(* IEC 61131-3 sources: SmartHomeNew/snapshots/2026-05-19 (part 4) *)

(* ---- FB_Water_Runtime_Hardening.st ---- *)
FUNCTION_BLOCK FB_Water_Runtime_Hardening
VAR_INPUT
    VI_Enable : BOOL;
    VI_System_Time_MS : UDINT;
END_VAR
VAR
    L_i : INT;

    L_FSM : ST_Water_Recovery_FSM_State;
    L_Event : ST_Water_Event_Log_Record;

    L_Empty_FSM : ST_Water_Recovery_FSM_State;
    L_Empty_Event : ST_Water_Event_Log_Record;

    L_Any_Rollback : BOOL;
    L_Any_Escalation : BOOL;
END_VAR

IF NOT VI_Enable THEN
    GVL_Water_Runtime_Hardening.G_Runtime_Valid := FALSE;
    RETURN;
END_IF;

L_Any_Rollback := FALSE;
L_Any_Escalation := FALSE;

FOR L_i := 1 TO GVL_CONSTANTS.C_MAX_FLOOD_SENSORS DO

    // Recovery FSM.
    L_FSM := L_Empty_FSM;
    L_FSM.Runtime_Valid := TRUE;

    L_FSM.Runtime_System_Time_MS :=
        VI_System_Time_MS;

    L_FSM.Recovery_Domain_Id :=
        GVL_Water_Topology_Config.G_Config_Record[L_i].Recovery_Domain_Id;

    L_FSM.Recovery_Requested :=
        GVL_INTENT_SAFETY.I_Water_Selective_Recovery_Allowed;

    L_FSM.Recovery_Sequencing_Active :=
        GVL_Water_Orchestration.G_Orchestration_State[L_i].Recovery_Sequence_Active;

    L_FSM.Recovery_Verification_Window_Active :=
        GVL_Water_Orchestration.G_Orchestration_State[L_i].Observation_Window_Active;

    // Conservative runtime hardening.
    IF GVL_Water_Physical_Runtime.G_Convergence_State[L_i].Escalation_Required THEN

        L_FSM.Rollback_Required := TRUE;
        L_FSM.Escalation_Required := TRUE;
        L_FSM.Operator_Ack_Required := TRUE;
        L_FSM.Recovery_Denied := TRUE;
        L_FSM.FSM_State := 100;

        L_FSM.Status_Code := 2;
        L_FSM.Status_Text :=
            'Recovery rollback escalation active';

    ELSIF L_FSM.Recovery_Requested THEN

        L_FSM.Recovery_Completed := TRUE;
        L_FSM.FSM_State := 10;

        L_FSM.Status_Code := 1;
        L_FSM.Status_Text :=
            'Recovery sequencing active';

    ELSE

        L_FSM.FSM_State := 0;

        L_FSM.Status_Code := 0;
        L_FSM.Status_Text :=
            'Recovery FSM idle';

    END_IF;

    GVL_Water_Runtime_Hardening.G_Recovery_FSM[L_i] :=
        L_FSM;

    // Runtime event publication.
    IF L_i <= 128 THEN

        L_Event := L_Empty_Event;
        L_Event.Runtime_Valid := TRUE;

        L_Event.Event_Time_MS := VI_System_Time_MS;
        L_Event.Event_Id := TO_UINT(L_i);

        IF L_FSM.Escalation_Required THEN
            L_Event.Event_Text :=
                'Water runtime escalation active';
        ELSE
            L_Event.Event_Text :=
                'Water runtime healthy';
        END_IF;

        GVL_Water_Runtime_Hardening.G_Event_Log[L_i] :=
            L_Event;

    END_IF;

    L_Any_Rollback :=
        L_Any_Rollback
        OR L_FSM.Rollback_Required;

    L_Any_Escalation :=
        L_Any_Escalation
        OR L_FSM.Escalation_Required;

END_FOR;

GVL_Water_Runtime_Hardening.G_Runtime_Quarantine_Active :=
    L_Any_Escalation;

GVL_Water_Runtime_Hardening.G_Service_Mode_Active := FALSE;
GVL_Water_Runtime_Hardening.G_Maintenance_Mode_Active := FALSE;

GVL_Water_Runtime_Hardening.G_Any_Rollback_Required :=
    L_Any_Rollback;

GVL_Water_Runtime_Hardening.G_Any_Escalation_Required :=
    L_Any_Escalation;

GVL_Water_Runtime_Hardening.G_Runtime_Valid := TRUE;
GVL_Water_Runtime_Hardening.G_Last_Update_MS := VI_System_Time_MS;

IF L_Any_Escalation THEN
    GVL_Water_Runtime_Hardening.G_Status_Code := 2;
    GVL_Water_Runtime_Hardening.G_Status_Text :=
        'Runtime quarantine escalation active';
ELSIF L_Any_Rollback THEN
    GVL_Water_Runtime_Hardening.G_Status_Code := 1;
    GVL_Water_Runtime_Hardening.G_Status_Text :=
        'Recovery rollback active';
ELSE
    GVL_Water_Runtime_Hardening.G_Status_Code := 0;
    GVL_Water_Runtime_Hardening.G_Status_Text :=
        'Production runtime hardening active';
END_IF;

END_FUNCTION_BLOCK

(* ---- FB_Water_Valve_Feedback_Runtime.st ---- *)
FUNCTION_BLOCK FB_Water_Valve_Feedback_Runtime
VAR_INPUT
    VI_Enable : BOOL;
    VI_System_Time_MS : UDINT;
END_VAR
VAR
    L_i : INT;

    L_Output : ST_Water_Output_Projection_State;
    L_State : ST_Water_Valve_Feedback_State;
    L_Empty_State : ST_Water_Valve_Feedback_State;

    L_Any_Degraded : BOOL;
    L_Any_Timeout : BOOL;
    L_Any_Conflict : BOOL;
END_VAR

IF NOT VI_Enable THEN
    GVL_Water_Valve_Feedback.G_Runtime_Valid := FALSE;
    RETURN;
END_IF;

L_Any_Degraded := FALSE;
L_Any_Timeout := FALSE;
L_Any_Conflict := FALSE;

FOR L_i := 1 TO GVL_CONSTANTS.C_MAX_FLOOD_SENSORS DO

    L_Output := GVL_Water_Output_Projection.G_Output_Projection_State[L_i];

    L_State := L_Empty_State;
    L_State.Runtime_Valid := TRUE;

    L_State.Runtime_System_Time_MS := VI_System_Time_MS;
    L_State.Valve_Group_Id := L_Output.Valve_Group_Id;

    // Feedback integration hook.
    // Conservative observe-only mode until physical DI binding is connected.
    L_State.Feedback_Available := FALSE;

    // No forced degraded state in observe-only mode.
    IF L_State.Feedback_Available THEN

        IF L_State.Physical_Open_Feedback
           AND L_State.Physical_Closed_Feedback THEN

            L_State.Feedback_Conflict := TRUE;
            L_State.Valve_Degraded := TRUE;

        END_IF;

        L_State.Confirmed_Open :=
            L_State.Physical_Open_Feedback
            AND NOT L_State.Physical_Closed_Feedback;

        L_State.Confirmed_Closed :=
            L_State.Physical_Closed_Feedback
            AND NOT L_State.Physical_Open_Feedback;

    ELSE

        L_State.Confirmation_Unknown := TRUE;

    END_IF;

    IF L_State.Feedback_Conflict THEN
        L_State.Status_Code := 3;
        L_State.Status_Text :=
            'Valve feedback conflict detected';
    ELSIF L_State.Feedback_Timeout THEN
        L_State.Status_Code := 2;
        L_State.Status_Text :=
            'Valve feedback timeout';
    ELSIF L_State.Confirmation_Unknown THEN
        L_State.Status_Code := 1;
        L_State.Status_Text :=
            'Valve feedback unavailable';
    ELSE
        L_State.Status_Code := 0;
        L_State.Status_Text :=
            'Valve feedback healthy';
    END_IF;

    GVL_Water_Valve_Feedback.G_Valve_Feedback_State[L_i] :=
        L_State;

    L_Any_Degraded :=
        L_Any_Degraded
        OR L_State.Valve_Degraded;

    L_Any_Timeout :=
        L_Any_Timeout
        OR L_State.Feedback_Timeout;

    L_Any_Conflict :=
        L_Any_Conflict
        OR L_State.Feedback_Conflict;

END_FOR;

GVL_Water_Valve_Feedback.G_Any_Degraded :=
    L_Any_Degraded;

GVL_Water_Valve_Feedback.G_Any_Timeout :=
    L_Any_Timeout;

GVL_Water_Valve_Feedback.G_Any_Conflict :=
    L_Any_Conflict;

GVL_Water_Valve_Feedback.G_Runtime_Valid := TRUE;
GVL_Water_Valve_Feedback.G_Last_Update_MS := VI_System_Time_MS;

IF L_Any_Conflict THEN
    GVL_Water_Valve_Feedback.G_Status_Code := 3;
    GVL_Water_Valve_Feedback.G_Status_Text :=
        'Valve feedback conflicts detected';
ELSIF L_Any_Timeout THEN
    GVL_Water_Valve_Feedback.G_Status_Code := 2;
    GVL_Water_Valve_Feedback.G_Status_Text :=
        'Valve feedback degraded';
ELSIF L_Any_Degraded THEN
    GVL_Water_Valve_Feedback.G_Status_Code := 1;
    GVL_Water_Valve_Feedback.G_Status_Text :=
        'Valve diagnostics degraded';
ELSE
    GVL_Water_Valve_Feedback.G_Status_Code := 0;
    GVL_Water_Valve_Feedback.G_Status_Text :=
        'Valve feedback runtime healthy';
END_IF;

END_FUNCTION_BLOCK

(* ---- FB_Water_Valve_Runtime_Governance.st ---- *)
FUNCTION_BLOCK FB_Water_Valve_Runtime_Governance
VAR_INPUT
    VI_Enable : BOOL;
    VI_System_Time_MS : UDINT;
END_VAR
VAR
    L_i : INT;

    L_Authority : ST_Water_Isolation_Authority_State;
    L_Valve : ST_Water_Valve_Runtime_State;
    L_Empty_Valve : ST_Water_Valve_Runtime_State;

    L_Any_Degraded : BOOL;
    L_Any_Confirmation_Unknown : BOOL;
    L_Any_Unsafe_Reopen : BOOL;
END_VAR

IF NOT VI_Enable THEN
    GVL_Water_Valve_Runtime.G_Runtime_Valid := FALSE;
    RETURN;
END_IF;

L_Any_Degraded := FALSE;
L_Any_Confirmation_Unknown := FALSE;
L_Any_Unsafe_Reopen := FALSE;

FOR L_i := 1 TO GVL_CONSTANTS.C_MAX_FLOOD_SENSORS DO

    L_Authority :=
        GVL_Water_Isolation_Authority.G_Authority_State[L_i];

    L_Valve := L_Empty_Valve;
    L_Valve.Runtime_Valid := TRUE;

    L_Valve.Runtime_System_Time_MS := VI_System_Time_MS;

    L_Valve.Valve_Id := L_Authority.Valve_Group_Id;
    L_Valve.Valve_Group_Id := L_Authority.Valve_Group_Id;

    L_Valve.Close_Requested :=
        L_Authority.Selective_Authority_Allowed
        OR L_Authority.Global_Fallback_Required;

    L_Valve.Global_Fallback_Request :=
        L_Authority.Global_Fallback_Required;

    L_Valve.Selective_Authority_Allowed :=
        L_Authority.Selective_Authority_Allowed;

    // Observe-only compatibility visibility.
    L_Valve.Physical_Output_Active :=
        GVL_COMMAND_SHADOW.G_Close_Valve_35
        OR GVL_COMMAND_SHADOW.G_Close_Valve_36;

    L_Valve.Output_Command_Projected :=
        L_Valve.Close_Requested;

    // Feedback/runtime hooks.
    L_Valve.Confirmation_Available :=
        GVL_Water_Valve_Feedback.G_Valve_Feedback_State[L_i].Feedback_Available;

    IF L_Valve.Confirmation_Available THEN

        L_Valve.Confirmed_Closed :=
            GVL_Water_Valve_Feedback.G_Valve_Feedback_State[L_i].Confirmed_Closed;

    ELSE

        L_Valve.Confirmation_Unknown := TRUE;

    END_IF;

    // Observe-only semantics must not force degraded state.
    L_Valve.Diagnostics_Available := FALSE;
    L_Valve.Valve_Healthy := TRUE;

    IF L_Valve.Confirmation_Available
       AND NOT L_Valve.Confirmed_Closed
       AND L_Valve.Close_Requested THEN

        L_Valve.Valve_Degraded := TRUE;

    END_IF;

    IF L_Valve.Valve_Degraded THEN

        L_Valve.Unsafe_Reopen_Denied := TRUE;
        L_Valve.Recovery_Allowed := FALSE;

        L_Valve.Status_Code := 2;
        L_Valve.Status_Text :=
            'Recovery denied: valve degraded';

    ELSIF L_Valve.Confirmation_Unknown THEN

        L_Valve.Status_Code := 1;
        L_Valve.Status_Text :=
            'Valve confirmation unavailable';

    ELSE

        L_Valve.Status_Code := 0;
        L_Valve.Status_Text :=
            'Valve governance runtime healthy';

    END_IF;

    GVL_Water_Valve_Runtime.G_Valve_Runtime_State[L_i] :=
        L_Valve;

    L_Any_Degraded :=
        L_Any_Degraded
        OR L_Valve.Valve_Degraded;

    L_Any_Confirmation_Unknown :=
        L_Any_Confirmation_Unknown
        OR L_Valve.Confirmation_Unknown;

    L_Any_Unsafe_Reopen :=
        L_Any_Unsafe_Reopen
        OR L_Valve.Unsafe_Reopen_Denied;

END_FOR;

GVL_Water_Valve_Runtime.G_Any_Valve_Degraded :=
    L_Any_Degraded;

GVL_Water_Valve_Runtime.G_Any_Confirmation_Unknown :=
    L_Any_Confirmation_Unknown;

GVL_Water_Valve_Runtime.G_Any_Unsafe_Reopen_Denied :=
    L_Any_Unsafe_Reopen;

GVL_Water_Valve_Runtime.G_Runtime_Valid := TRUE;
GVL_Water_Valve_Runtime.G_Last_Update_MS := VI_System_Time_MS;

IF L_Any_Degraded THEN
    GVL_Water_Valve_Runtime.G_Status_Code := 2;
    GVL_Water_Valve_Runtime.G_Status_Text :=
        'Valve governance degraded';
ELSIF L_Any_Confirmation_Unknown THEN
    GVL_Water_Valve_Runtime.G_Status_Code := 1;
    GVL_Water_Valve_Runtime.G_Status_Text :=
        'Valve confirmation unknown';
ELSE
    GVL_Water_Valve_Runtime.G_Status_Code := 0;
    GVL_Water_Valve_Runtime.G_Status_Text :=
        'Valve governance runtime active';
END_IF;

END_FUNCTION_BLOCK

(* ---- PRG_Authority_Provenance_Governor.st ---- *)
PROGRAM PRG_Authority_Provenance_Governor
VAR
    L_Now_MS : UDINT;
    L_Provenance_Valid : BOOL := TRUE;
    L_Error_Code : UDINT := 0;
    L_Error_Text : STRING(160) := '';
END_VAR

L_Now_MS := GVL_STATUS.G_System_Time_MS;
L_Provenance_Valid := TRUE;
L_Error_Code := 0;
L_Error_Text := '';

// Fail-safe defaults.
GVL_AUTHORITY_PROVENANCE_FABRIC.Authority_Provenance_Valid := FALSE;
GVL_AUTHORITY_PROVENANCE_FABRIC.Authority_Provenance_Granted := FALSE;
GVL_AUTHORITY_PROVENANCE_FABRIC.Authority_Provenance_Quarantine_Active := TRUE;

GVL_AUTHORITY_PROVENANCE_FABRIC.Bootstrap_Authority_Authentic := FALSE;
GVL_AUTHORITY_PROVENANCE_FABRIC.Commissioning_Lineage_Traceable := FALSE;
GVL_AUTHORITY_PROVENANCE_FABRIC.Trust_Seed_Integrity_Valid := FALSE;
GVL_AUTHORITY_PROVENANCE_FABRIC.Root_Authority_Attribution_Coherent := FALSE;
GVL_AUTHORITY_PROVENANCE_FABRIC.Provenance_Causality_Grounded := FALSE;

// Meta-governance required.
IF NOT GVL_META_GOVERNANCE_FABRIC.Meta_Governance_Granted THEN
    L_Provenance_Valid := FALSE;
    L_Error_Code := 46000;
    L_Error_Text := 'Meta-governance authority not granted';
END_IF;

// Authority-origin split-brain detectors.
IF GVL_AUTHORITY_PROVENANCE_FABRIC.Bootstrap_Identity_Corruption_Detected THEN
    L_Provenance_Valid := FALSE;
    L_Error_Code := 46001;
    L_Error_Text := 'Bootstrap identity corruption detected';
END_IF;

IF GVL_AUTHORITY_PROVENANCE_FABRIC.Forged_Authority_Root_Detected THEN
    L_Provenance_Valid := FALSE;
    L_Error_Code := 46002;
    L_Error_Text := 'Forged authority root detected';
END_IF;

IF GVL_AUTHORITY_PROVENANCE_FABRIC.Commissioning_Provenance_Gap_Detected THEN
    L_Provenance_Valid := FALSE;
    L_Error_Code := 46003;
    L_Error_Text := 'Commissioning provenance gap detected';
END_IF;

IF GVL_AUTHORITY_PROVENANCE_FABRIC.Trust_Seed_Impersonation_Detected THEN
    L_Provenance_Valid := FALSE;
    L_Error_Code := 46004;
    L_Error_Text := 'Trust seed impersonation detected';
END_IF;

IF GVL_AUTHORITY_PROVENANCE_FABRIC.Origin_Authenticity_Erosion_Detected THEN
    L_Provenance_Valid := FALSE;
    L_Error_Code := 46005;
    L_Error_Text := 'Origin authenticity erosion detected';
END_IF;

IF GVL_AUTHORITY_PROVENANCE_FABRIC.Root_Lineage_Tampering_Detected THEN
    L_Provenance_Valid := FALSE;
    L_Error_Code := 46006;
    L_Error_Text := 'Root lineage tampering detected';
END_IF;

// Provenance integrity validation.
IF L_Provenance_Valid
AND NOT GVL_AUTHORITY_PROVENANCE_FABRIC.Historical_Origin_Lineage_Valid THEN
    L_Provenance_Valid := FALSE;
    L_Error_Code := 46010;
    L_Error_Text := 'Historical origin lineage invalid';
END_IF;

IF L_Provenance_Valid
AND NOT GVL_AUTHORITY_PROVENANCE_FABRIC.Distributed_Trust_Chain_Coherent THEN
    L_Provenance_Valid := FALSE;
    L_Error_Code := 46011;
    L_Error_Text := 'Distributed trust chain coherence invalid';
END_IF;

IF L_Provenance_Valid
AND NOT GVL_AUTHORITY_PROVENANCE_FABRIC.Authority_Origin_Continuity_Stable THEN
    L_Provenance_Valid := FALSE;
    L_Error_Code := 46012;
    L_Error_Text := 'Authority origin continuity invalid';
END_IF;

IF L_Provenance_Valid
AND NOT GVL_AUTHORITY_PROVENANCE_FABRIC.Root_Identity_Cryptographic_Validity THEN
    L_Provenance_Valid := FALSE;
    L_Error_Code := 46013;
    L_Error_Text := 'Root identity cryptographic validity invalid';
END_IF;

IF L_Provenance_Valid THEN
    GVL_AUTHORITY_PROVENANCE_FABRIC.Authority_Provenance_Valid := TRUE;
    GVL_AUTHORITY_PROVENANCE_FABRIC.Authority_Provenance_Granted := TRUE;
    GVL_AUTHORITY_PROVENANCE_FABRIC.Authority_Provenance_Quarantine_Active := FALSE;

    GVL_AUTHORITY_PROVENANCE_FABRIC.Bootstrap_Authority_Authentic := TRUE;
    GVL_AUTHORITY_PROVENANCE_FABRIC.Commissioning_Lineage_Traceable := TRUE;
    GVL_AUTHORITY_PROVENANCE_FABRIC.Trust_Seed_Integrity_Valid := TRUE;
    GVL_AUTHORITY_PROVENANCE_FABRIC.Root_Authority_Attribution_Coherent := TRUE;
    GVL_AUTHORITY_PROVENANCE_FABRIC.Provenance_Causality_Grounded := TRUE;

    GVL_AUTHORITY_PROVENANCE_FABRIC.Authority_Provenance_Epoch :=
        GVL_META_GOVERNANCE_FABRIC.Meta_Governance_Epoch;

    GVL_AUTHORITY_PROVENANCE_FABRIC.Authority_Provenance_Epoch_Coherent := TRUE;

    GVL_AUTHORITY_PROVENANCE_FABRIC.Authority_Provenance_Last_Update_MS :=
        L_Now_MS;

    GVL_AUTHORITY_PROVENANCE_FABRIC.Authority_Provenance_Lease_Expired := FALSE;

    GVL_AUTHORITY_PROVENANCE_FABRIC.Authority_Provenance_Last_Error_Code := 0;
    GVL_AUTHORITY_PROVENANCE_FABRIC.Authority_Provenance_Last_Error_Text := '';
ELSE
    GVL_AUTHORITY_PROVENANCE_FABRIC.Authority_Provenance_Valid := FALSE;
    GVL_AUTHORITY_PROVENANCE_FABRIC.Authority_Provenance_Granted := FALSE;
    GVL_AUTHORITY_PROVENANCE_FABRIC.Authority_Provenance_Quarantine_Active := TRUE;

    GVL_AUTHORITY_PROVENANCE_FABRIC.Authority_Provenance_Lease_Expired := TRUE;

    GVL_AUTHORITY_PROVENANCE_FABRIC.Authority_Provenance_Last_Error_Code :=
        L_Error_Code;

    GVL_AUTHORITY_PROVENANCE_FABRIC.Authority_Provenance_Last_Error_Text :=
        L_Error_Text;

    GVL_AUTHORITY_PROVENANCE_FABRIC.Authority_Provenance_Invalidation_Count :=
        GVL_AUTHORITY_PROVENANCE_FABRIC.Authority_Provenance_Invalidation_Count + 1;
END_IF;

END_PROGRAM

(* ---- PRG_Authority_Restoration_Governor.st ---- *)
PROGRAM PRG_Authority_Restoration_Governor
VAR
    L_Now_MS : UDINT;
    L_Restoration_Valid : BOOL := TRUE;
END_VAR

L_Now_MS := GVL_STATUS.G_System_Time_MS;
L_Restoration_Valid := TRUE;

// Fail-safe defaults.
GVL_AUTHORITY_RESTORATION.Authority_Restoration_Active := FALSE;
GVL_AUTHORITY_RESTORATION.Authority_Restoration_Allowed := FALSE;
GVL_AUTHORITY_RESTORATION.Authority_Restoration_Completed := FALSE;

GVL_AUTHORITY_RESTORATION.Snapshot_Restoration_Valid := FALSE;
GVL_AUTHORITY_RESTORATION.Consensus_Restoration_Valid := FALSE;
GVL_AUTHORITY_RESTORATION.Causality_Restoration_Valid := FALSE;
GVL_AUTHORITY_RESTORATION.Epoch_Restoration_Valid := FALSE;
GVL_AUTHORITY_RESTORATION.Lineage_Restoration_Valid := FALSE;

GVL_AUTHORITY_RESTORATION.Revocation_Clearance_Valid := FALSE;
GVL_AUTHORITY_RESTORATION.Stabilization_Window_Elapsed := FALSE;
GVL_AUTHORITY_RESTORATION.Reauthorization_Order_Valid := FALSE;

// Restoration impossible while revocation active.
IF GVL_AUTHORITY_REVOCATION.Authority_Revocation_Active THEN
    L_Restoration_Valid := FALSE;
END_IF;

// Snapshot must recover first.
IF L_Restoration_Valid
AND NOT GVL_PHYSICAL_SNAPSHOT.Physical_Snapshot_Valid THEN
    L_Restoration_Valid := FALSE;
END_IF;

IF L_Restoration_Valid THEN
    GVL_AUTHORITY_RESTORATION.Snapshot_Restoration_Valid := TRUE;
END_IF;

// Consensus recovery.
IF L_Restoration_Valid
AND NOT GVL_SENSOR_CONSENSUS.Sensor_Consensus_Valid THEN
    L_Restoration_Valid := FALSE;
END_IF;

IF L_Restoration_Valid THEN
    GVL_AUTHORITY_RESTORATION.Consensus_Restoration_Valid := TRUE;
END_IF;

// Telemetry causality recovery.
IF L_Restoration_Valid
AND NOT GVL_TELEMETRY.Command_Telemetry_Causality_Valid THEN
    L_Restoration_Valid := FALSE;
END_IF;

IF L_Restoration_Valid THEN
    GVL_AUTHORITY_RESTORATION.Causality_Restoration_Valid := TRUE;
END_IF;

// Epoch coherence recovery.
IF L_Restoration_Valid
AND NOT GVL_PHYSICAL_AUTHORITY_EPOCH.Physical_Authority_Epoch_Valid THEN
    L_Restoration_Valid := FALSE;
END_IF;

IF L_Restoration_Valid THEN
    GVL_AUTHORITY_RESTORATION.Epoch_Restoration_Valid := TRUE;
END_IF;

// Lineage continuity recovery.
IF L_Restoration_Valid
AND NOT GVL_AUTHORITY_LINEAGE.Authority_Lineage_Valid THEN
    L_Restoration_Valid := FALSE;
END_IF;

IF L_Restoration_Valid THEN
    GVL_AUTHORITY_RESTORATION.Lineage_Restoration_Valid := TRUE;
END_IF;

// Revocation must be fully cleared.
IF L_Restoration_Valid
AND GVL_AUTHORITY_REVOCATION.Quarantine_Fabric_Active THEN
    L_Restoration_Valid := FALSE;
END_IF;

IF L_Restoration_Valid THEN
    GVL_AUTHORITY_RESTORATION.Revocation_Clearance_Valid := TRUE;
END_IF;

// Stabilization window after recovery.
IF L_Restoration_Valid
AND ((L_Now_MS - GVL_AUTHORITY_REVOCATION.Revocation_Last_Update_MS) < 5000) THEN
    L_Restoration_Valid := FALSE;
END_IF;

IF L_Restoration_Valid THEN
    GVL_AUTHORITY_RESTORATION.Stabilization_Window_Elapsed := TRUE;
END_IF;

IF L_Restoration_Valid THEN
    GVL_AUTHORITY_RESTORATION.Authority_Restoration_Active := TRUE;
    GVL_AUTHORITY_RESTORATION.Authority_Restoration_Allowed := TRUE;
    GVL_AUTHORITY_RESTORATION.Authority_Restoration_Completed := TRUE;

    GVL_AUTHORITY_RESTORATION.Reauthorization_Order_Valid := TRUE;

    GVL_AUTHORITY_RESTORATION.Restoration_Epoch :=
        GVL_PHYSICAL_AUTHORITY_EPOCH.Physical_Authority_Epoch;

    GVL_AUTHORITY_RESTORATION.Restoration_Last_Update_MS := L_Now_MS;
END_IF;

END_PROGRAM

(* ---- PRG_Command_Arbitration.st ---- *)
PROGRAM PRG_Command_Arbitration
VAR
    L_Mode : E_Safety_Mode;
    L_Safety_Active : BOOL;
    L_User_Access_OK : BOOL;
    L_i : INT;

    // Local deterministic command buffer
    L_Gas_Valve_Close : BOOL;
    L_Boiler_Stop : BOOL;
    L_Supply_100_Req : BOOL;
    L_Supply_80_Req : BOOL;
    L_Vent_PV3_Boost : BOOL;
    L_Exhaust_100_Req : BOOL;
    L_Vent_Stop : BOOL;
    L_Vent_Block : BOOL;
    L_Vent_Smoke_Exhaust : BOOL;

    L_Heating_Block : BOOL;
    L_Heating_Emergency_Stop : BOOL;
    L_Heating_Gas_Safety_Stop : BOOL;

    L_Water_Block : BOOL;
    L_Water_Emergency_Stop : BOOL;
    L_Close_Valve_35 : BOOL;
    L_Close_Valve_36 : BOOL;

    L_Lock_1_Open : BOOL;
    L_Lock_1_Close : BOOL;
    L_Lock_2_Open : BOOL;
    L_Lock_2_Close : BOOL;
    L_Gate_Open : BOOL;
    L_Wicket_Open : BOOL;
END_VAR

// ======================================================
// PRIORITY 1: PLC ROLE VALIDATION (ABSOLUTE)
// ======================================================
IF GVL_STATUS.G_Is_Active_PLC AND GVL_STATUS.G_Other_PLC_Is_Active THEN
    GVL_HEALTH_BRIDGE.G_Role_Conflict_Error := TRUE;

    GVL_COMMAND_SHADOW.G_Gas_Valve_Close := TRUE;
    GVL_COMMAND_SHADOW.G_Boiler_Stop := TRUE;
    GVL_COMMAND_SHADOW.G_Supply_100_Req := FALSE;
    GVL_COMMAND_SHADOW.G_Supply_80_Req := FALSE;
    GVL_COMMAND_SHADOW.G_Vent_PV3_Boost := FALSE;
    GVL_COMMAND_SHADOW.G_Exhaust_100_Req := FALSE;
    GVL_COMMAND_SHADOW.G_Vent_Stop := TRUE;
    GVL_COMMAND_SHADOW.G_Vent_Block := TRUE;
    GVL_COMMAND_SHADOW.G_Vent_Smoke_Exhaust := FALSE;

    GVL_COMMAND_SHADOW.G_Heating_Block := TRUE;
    GVL_COMMAND_SHADOW.G_Heating_Emergency_Stop := TRUE;
    GVL_COMMAND_SHADOW.G_Heating_Gas_Safety_Stop := TRUE;

    GVL_COMMAND_SHADOW.G_Water_Block := TRUE;
    GVL_COMMAND_SHADOW.G_Water_Emergency_Stop := TRUE;
    GVL_COMMAND_SHADOW.G_Close_Valve_35 := TRUE;
    GVL_COMMAND_SHADOW.G_Close_Valve_36 := TRUE;

    GVL_COMMAND_SHADOW.G_Lock_1_Open := FALSE;
    GVL_COMMAND_SHADOW.G_Lock_1_Close := FALSE;
    GVL_COMMAND_SHADOW.G_Lock_2_Open := FALSE;
    GVL_COMMAND_SHADOW.G_Lock_2_Close := FALSE;
    GVL_COMMAND_SHADOW.G_Gate_Open := FALSE;
    GVL_COMMAND_SHADOW.G_Wicket_Open := FALSE;
    RETURN;
END_IF;

// ======================================================
// PRIORITY 2: PLC INACTIVE
// ======================================================
IF NOT GVL_STATUS.G_Is_Active_PLC THEN
    GVL_COMMAND_SHADOW.G_Gas_Valve_Close := GVL_COMMAND_POLICY_CONFIG.G_PLC_Inactive_Close_Gas;
    GVL_COMMAND_SHADOW.G_Boiler_Stop := GVL_COMMAND_POLICY_CONFIG.G_PLC_Inactive_Stop_Boiler;
    GVL_COMMAND_SHADOW.G_Supply_100_Req := FALSE;
    GVL_COMMAND_SHADOW.G_Supply_80_Req := FALSE;
    GVL_COMMAND_SHADOW.G_Vent_PV3_Boost := FALSE;
    GVL_COMMAND_SHADOW.G_Exhaust_100_Req := FALSE;
    GVL_COMMAND_SHADOW.G_Vent_Stop := GVL_COMMAND_POLICY_CONFIG.G_PLC_Inactive_Stop_Vent;
    GVL_COMMAND_SHADOW.G_Vent_Block := FALSE;
    GVL_COMMAND_SHADOW.G_Vent_Smoke_Exhaust := FALSE;

    GVL_COMMAND_SHADOW.G_Heating_Block := GVL_COMMAND_POLICY_CONFIG.G_PLC_Inactive_Block_Heating;
    GVL_COMMAND_SHADOW.G_Heating_Emergency_Stop := FALSE;
    GVL_COMMAND_SHADOW.G_Heating_Gas_Safety_Stop := FALSE;

    GVL_COMMAND_SHADOW.G_Water_Block := GVL_COMMAND_POLICY_CONFIG.G_PLC_Inactive_Block_Water;
    GVL_COMMAND_SHADOW.G_Water_Emergency_Stop := FALSE;
    GVL_COMMAND_SHADOW.G_Close_Valve_35 := FALSE;
    GVL_COMMAND_SHADOW.G_Close_Valve_36 := FALSE;

    GVL_COMMAND_SHADOW.G_Lock_1_Open := FALSE;
    GVL_COMMAND_SHADOW.G_Lock_1_Close := FALSE;
    GVL_COMMAND_SHADOW.G_Lock_2_Open := FALSE;
    GVL_COMMAND_SHADOW.G_Lock_2_Close := FALSE;
    GVL_COMMAND_SHADOW.G_Gate_Open := FALSE;
    GVL_COMMAND_SHADOW.G_Wicket_Open := FALSE;
    RETURN;
END_IF;

// ======================================================
// RESET LOCAL BUFFER
// ======================================================
L_Gas_Valve_Close := FALSE;
L_Boiler_Stop := FALSE;
L_Supply_100_Req := FALSE;
L_Supply_80_Req := FALSE;
L_Vent_PV3_Boost := FALSE;
L_Exhaust_100_Req := FALSE;
L_Vent_Stop := FALSE;
L_Vent_Block := FALSE;
L_Vent_Smoke_Exhaust := FALSE;

L_Heating_Block := FALSE;
L_Heating_Emergency_Stop := FALSE;
L_Heating_Gas_Safety_Stop := FALSE;

L_Water_Block := FALSE;
L_Water_Emergency_Stop := FALSE;
L_Close_Valve_35 := FALSE;
L_Close_Valve_36 := FALSE;

L_Lock_1_Open := FALSE;
L_Lock_1_Close := FALSE;
L_Lock_2_Open := FALSE;
L_Lock_2_Close := FALSE;
L_Gate_Open := FALSE;
L_Wicket_Open := FALSE;

// ======================================================
// PRIORITY 3: SAFETY MODE
// ======================================================
L_Mode := GVL_SAFETY_SHUTDOWN.G_Safety_Mode;
L_Safety_Active := FALSE;

CASE L_Mode OF

    NORMAL:
        L_Safety_Active := FALSE;

    FIRE:
        L_Safety_Active := TRUE;
        L_Heating_Block := GVL_COMMAND_POLICY_CONFIG.G_Fire_Block_Heating;
        L_Boiler_Stop := GVL_COMMAND_POLICY_CONFIG.G_Fire_Stop_Boiler;
        L_Vent_Stop := FALSE;
        L_Vent_PV3_Boost := FALSE;
        L_Exhaust_100_Req := FALSE;
        L_Vent_Smoke_Exhaust := TRUE;
        L_Heating_Emergency_Stop := GVL_COMMAND_POLICY_CONFIG.G_Fire_Block_Heating;
        L_Lock_1_Open := GVL_COMMAND_POLICY_CONFIG.G_Fire_Open_Lock_1;
        L_Lock_2_Open := GVL_COMMAND_POLICY_CONFIG.G_Fire_Open_Lock_2;
        L_Gate_Open := GVL_COMMAND_POLICY_CONFIG.G_Fire_Open_Gate;
        L_Wicket_Open := GVL_COMMAND_POLICY_CONFIG.G_Fire_Open_Wicket;

    GAS:
        L_Safety_Active := TRUE;
        L_Gas_Valve_Close := GVL_COMMAND_POLICY_CONFIG.G_Gas_Close_Gas;
        L_Boiler_Stop := GVL_COMMAND_POLICY_CONFIG.G_Gas_Stop_Boiler;
        L_Heating_Block := GVL_COMMAND_POLICY_CONFIG.G_Gas_Block_Heating;
        L_Heating_Gas_Safety_Stop := GVL_COMMAND_POLICY_CONFIG.G_Gas_Block_Heating;
        L_Vent_PV3_Boost := TRUE;
        L_Vent_Smoke_Exhaust := FALSE;
        L_Gate_Open := GVL_COMMAND_POLICY_CONFIG.G_Gas_Open_Gate;
        L_Wicket_Open := GVL_COMMAND_POLICY_CONFIG.G_Gas_Open_Wicket;
        L_Lock_1_Open := GVL_COMMAND_POLICY_CONFIG.G_Gas_Open_Lock_1;
        L_Lock_2_Open := GVL_COMMAND_POLICY_CONFIG.G_Gas_Open_Lock_2;

    WATER_LEAK:
        L_Safety_Active := TRUE;
        L_Water_Block := GVL_COMMAND_POLICY_CONFIG.G_Water_Block_Water;
        L_Water_Emergency_Stop := GVL_COMMAND_POLICY_CONFIG.G_Water_Block_Water;
        L_Close_Valve_35 := GVL_COMMAND_POLICY_CONFIG.G_Water_Block_Water;
        L_Close_Valve_36 := GVL_COMMAND_POLICY_CONFIG.G_Water_Block_Water;

    GLOBAL_STOP:
        L_Safety_Active := TRUE;
        L_Heating_Block := GVL_COMMAND_POLICY_CONFIG.G_GlobalStop_Block_Heating;
        L_Heating_Emergency_Stop := GVL_COMMAND_POLICY_CONFIG.G_GlobalStop_Block_Heating;
        L_Boiler_Stop := GVL_COMMAND_POLICY_CONFIG.G_GlobalStop_Stop_Boiler;
        L_Vent_Stop := GVL_COMMAND_POLICY_CONFIG.G_GlobalStop_Stop_Vent;
        L_Water_Block := GVL_COMMAND_POLICY_CONFIG.G_GlobalStop_Block_Water;
        L_Water_Emergency_Stop := GVL_COMMAND_POLICY_CONFIG.G_GlobalStop_Block_Water;
        L_Close_Valve_35 := GVL_COMMAND_POLICY_CONFIG.G_GlobalStop_Block_Water;
        L_Close_Valve_36 := GVL_COMMAND_POLICY_CONFIG.G_GlobalStop_Block_Water;

ELSE
        L_Safety_Active := TRUE;
        L_Gas_Valve_Close := TRUE;
        L_Boiler_Stop := TRUE;
        L_Heating_Block := TRUE;
        L_Heating_Emergency_Stop := TRUE;
        L_Vent_Stop := TRUE;
        L_Water_Block := TRUE;
        L_Water_Emergency_Stop := TRUE;
        L_Close_Valve_35 := TRUE;
        L_Close_Valve_36 := TRUE;
END_CASE;

// ======================================================
// PRIORITY 4: USER INTENT (ONLY WHEN SAFETY IS NOT ACTIVE)
// ======================================================
L_User_Access_OK := GVL_INTENT_USER.I_Source_Valid AND (GVL_INTENT_USER.I_User_Access_Level >= 1);

IF (NOT L_Safety_Active) AND L_User_Access_OK THEN
    IF GVL_INTENT_USER.I_Lock_1_Open_Request THEN
        L_Lock_1_Open := TRUE;
        L_Lock_1_Close := FALSE;
    ELSIF GVL_INTENT_USER.I_Lock_1_Close_Request THEN
        L_Lock_1_Open := FALSE;
        L_Lock_1_Close := TRUE;
    END_IF;

    IF GVL_INTENT_USER.I_Lock_2_Open_Request THEN
        L_Lock_2_Open := TRUE;
        L_Lock_2_Close := FALSE;
    ELSIF GVL_INTENT_USER.I_Lock_2_Close_Request THEN
        L_Lock_2_Open := FALSE;
        L_Lock_2_Close := TRUE;
    END_IF;

    IF GVL_INTENT_USER.I_Gate_Open_Request THEN
        L_Gate_Open := TRUE;
    END_IF;

    IF GVL_INTENT_USER.I_Wicket_Open_Request THEN
        L_Wicket_Open := TRUE;
    END_IF;
END_IF;

// Dangerous user actions require explicit confirmation and elevated access.
IF (NOT L_Safety_Active) AND
   GVL_INTENT_USER.I_Source_Valid AND
   GVL_INTENT_USER.I_Dangerous_Action_Request AND
   GVL_INTENT_USER.I_Dangerous_Action_Confirm AND
   (GVL_INTENT_USER.I_User_Access_Level >= 2) THEN
    // Reserved for future high-risk manual actions.
    // No direct safety override is allowed here.
END_IF;

// ======================================================
// PRIORITY 5: AUTOMATION RULES (ONLY SAFE COMMAND-LEVEL ACTIONS)
// ======================================================
IF NOT L_Safety_Active THEN
    FOR L_i := 1 TO GVL_CONSTANTS.C_MAX_RULES DO
        IF GVL_STATE.G_Rule_Actions[L_i].Active AND GVL_STATE.G_Rule_Actions[L_i].Triggered THEN
            CASE GVL_STATE.G_Rule_Actions[L_i].Action_Type OF

                ACTION_SET_FLOOR_HEATING:
                    IF GVL_STATE.G_Rule_Actions[L_i].Value <= 0.0 THEN
                        L_Heating_Block := TRUE;
                        L_Boiler_Stop := TRUE;
                    END_IF;

                ACTION_SET_VENTILATION:
                    IF GVL_STATE.G_Rule_Actions[L_i].Value <= 0.0 THEN
                        L_Vent_Stop := TRUE;
                    END_IF;

            ELSE
                // Non command-level actions are handled by their own subsystem.
            END_CASE;
        END_IF;
    END_FOR;
END_IF;

// ======================================================
// POST-PROCESS CONFLICT RESOLUTION
// ======================================================
IF (L_Mode = FIRE) AND GVL_COMMAND_POLICY_CONFIG.G_Fire_Block_Lock_Close THEN
    L_Lock_1_Close := FALSE;
    L_Lock_2_Close := FALSE;
END_IF;

IF GVL_COMMAND_POLICY_CONFIG.G_Block_Close_When_Open_Commanded THEN
    IF L_Lock_1_Open AND L_Lock_1_Close THEN
        L_Lock_1_Close := FALSE;
    END_IF;

    IF L_Lock_2_Open AND L_Lock_2_Close THEN
        L_Lock_2_Close := FALSE;
    END_IF;
END_IF;

// ======================================================
// SINGLE POINT WRITE (DETERMINISTIC)
// ======================================================
GVL_COMMAND_SHADOW.G_Gas_Valve_Close := L_Gas_Valve_Close;
GVL_COMMAND_SHADOW.G_Boiler_Stop := L_Boiler_Stop;
GVL_COMMAND_SHADOW.G_Supply_100_Req := L_Supply_100_Req;
GVL_COMMAND_SHADOW.G_Supply_80_Req := L_Supply_80_Req;
GVL_COMMAND_SHADOW.G_Vent_PV3_Boost := L_Vent_PV3_Boost;
GVL_COMMAND_SHADOW.G_Exhaust_100_Req := L_Exhaust_100_Req;
GVL_COMMAND_SHADOW.G_Vent_Stop := L_Vent_Stop;
GVL_COMMAND_SHADOW.G_Vent_Block := L_Vent_Block;
GVL_COMMAND_SHADOW.G_Vent_Smoke_Exhaust := L_Vent_Smoke_Exhaust;

GVL_COMMAND_SHADOW.G_Heating_Block := L_Heating_Block;
GVL_COMMAND_SHADOW.G_Heating_Emergency_Stop := L_Heating_Emergency_Stop;
GVL_COMMAND_SHADOW.G_Heating_Gas_Safety_Stop := L_Heating_Gas_Safety_Stop;

GVL_COMMAND_SHADOW.G_Water_Block := L_Water_Block;
GVL_COMMAND_SHADOW.G_Water_Emergency_Stop := L_Water_Emergency_Stop;
GVL_COMMAND_SHADOW.G_Close_Valve_35 := L_Close_Valve_35;
GVL_COMMAND_SHADOW.G_Close_Valve_36 := L_Close_Valve_36;

GVL_COMMAND_SHADOW.G_Lock_1_Open := L_Lock_1_Open;
GVL_COMMAND_SHADOW.G_Lock_1_Close := L_Lock_1_Close;
GVL_COMMAND_SHADOW.G_Lock_2_Open := L_Lock_2_Open;
GVL_COMMAND_SHADOW.G_Lock_2_Close := L_Lock_2_Close;
GVL_COMMAND_SHADOW.G_Gate_Open := L_Gate_Open;
GVL_COMMAND_SHADOW.G_Wicket_Open := L_Wicket_Open;

// >>> BULK_SYNC_ANCHOR: PRG_Command_Arbitration <<<
END_PROGRAM

(* ---- PRG_Command_Verifier.st ---- *)
PROGRAM PRG_Command_Verifier
VAR
    L_i : INT;
    L_Mismatch_Count : INT := 0;
    L_Runtime_Error : BOOL := FALSE;
    L_Runtime_Error_Code : UDINT := 0;
    L_Runtime_Error_Text : STRING(160) := '';
    L_Now_MS : UDINT;
    L_Prev_Runtime_Error : BOOL;
    L_Any_Manifold_Pump_On : BOOL;
    fbLog : FB_LogEvent;
END_VAR

L_Now_MS := GVL_STATUS.G_System_Time_MS;

// ===============================
// 1. COMMAND MISMATCH CHECK
// ===============================
L_Mismatch_Count := 0;

IF GVL_COMMAND.G_Gas_Valve_Close <> GVL_COMMAND_SHADOW.G_Gas_Valve_Close THEN L_Mismatch_Count := L_Mismatch_Count + 1; END_IF;
IF GVL_COMMAND.G_Boiler_Stop <> GVL_COMMAND_SHADOW.G_Boiler_Stop THEN L_Mismatch_Count := L_Mismatch_Count + 1; END_IF;
IF GVL_COMMAND.G_Vent_Stop <> GVL_COMMAND_SHADOW.G_Vent_Stop THEN L_Mismatch_Count := L_Mismatch_Count + 1; END_IF;
IF GVL_COMMAND.G_Supply_100_Req <> GVL_COMMAND_SHADOW.G_Supply_100_Req THEN L_Mismatch_Count := L_Mismatch_Count + 1; END_IF;
IF GVL_COMMAND.G_Supply_80_Req <> GVL_COMMAND_SHADOW.G_Supply_80_Req THEN L_Mismatch_Count := L_Mismatch_Count + 1; END_IF;
IF GVL_COMMAND.G_Vent_PV3_Boost <> GVL_COMMAND_SHADOW.G_Vent_PV3_Boost THEN L_Mismatch_Count := L_Mismatch_Count + 1; END_IF;
IF GVL_COMMAND.G_Close_Valve_35 <> GVL_COMMAND_SHADOW.G_Close_Valve_35 THEN L_Mismatch_Count := L_Mismatch_Count + 1; END_IF;
IF GVL_COMMAND.G_Close_Valve_36 <> GVL_COMMAND_SHADOW.G_Close_Valve_36 THEN L_Mismatch_Count := L_Mismatch_Count + 1; END_IF;
IF GVL_COMMAND.G_Lock_1_Open <> GVL_COMMAND_SHADOW.G_Lock_1_Open THEN L_Mismatch_Count := L_Mismatch_Count + 1; END_IF;
IF GVL_COMMAND.G_Lock_1_Close <> GVL_COMMAND_SHADOW.G_Lock_1_Close THEN L_Mismatch_Count := L_Mismatch_Count + 1; END_IF;
IF GVL_COMMAND.G_Lock_2_Open <> GVL_COMMAND_SHADOW.G_Lock_2_Open THEN L_Mismatch_Count := L_Mismatch_Count + 1; END_IF;
IF GVL_COMMAND.G_Lock_2_Close <> GVL_COMMAND_SHADOW.G_Lock_2_Close THEN L_Mismatch_Count := L_Mismatch_Count + 1; END_IF;
IF GVL_COMMAND.G_Gate_Open <> GVL_COMMAND_SHADOW.G_Gate_Open THEN L_Mismatch_Count := L_Mismatch_Count + 1; END_IF;
IF GVL_COMMAND.G_Wicket_Open <> GVL_COMMAND_SHADOW.G_Wicket_Open THEN L_Mismatch_Count := L_Mismatch_Count + 1; END_IF;

GVL_COMMAND_VERIFY.Command_Mismatch_Count := L_Mismatch_Count;
GVL_COMMAND_VERIFY.Command_Match_OK := (L_Mismatch_Count = 0);
GVL_COMMAND_VERIFY.Command_Mismatch_Active := (L_Mismatch_Count > 0);

// ===============================
// 2. RUNTIME SANITY CHECKS
// ===============================
L_Runtime_Error := FALSE;
L_Runtime_Error_Code := 0;
L_Runtime_Error_Text := '';
L_Any_Manifold_Pump_On := FALSE;

// PLC inactive: fail-safe outputs should be off/safe except alarm/gas close outputs.
IF (NOT L_Runtime_Error) AND (NOT GVL_STATUS.G_Is_Active_PLC) THEN
    FOR L_i := 1 TO GVL_CONSTANTS.C_MAX_HEATING_CIRCUITS DO
        IF GVL_IO.DO_Zone_Valves[L_i] THEN
            L_Runtime_Error := TRUE;
            L_Runtime_Error_Code := 10;
            L_Runtime_Error_Text := 'PLC inactive zone valve on';
        END_IF;
    END_FOR;
END_IF;

IF (NOT L_Runtime_Error) AND (NOT GVL_STATUS.G_Is_Active_PLC) THEN
    FOR L_i := 1 TO GVL_CONSTANTS.C_MAX_MANIFOLDS DO
        IF GVL_IO.DO_Manifold_Pumps[L_i] THEN
            L_Runtime_Error := TRUE;
            L_Runtime_Error_Code := 11;
            L_Runtime_Error_Text := 'PLC inactive pump on';
        END_IF;
    END_FOR;
END_IF;

// GAS: gas valve must be physically commanded closed.
IF (NOT L_Runtime_Error) AND (GVL_SAFETY_SHUTDOWN.G_Safety_Mode = GAS) AND (NOT GVL_IO.DO_Gas_Valve_Close) THEN
    L_Runtime_Error := TRUE;
    L_Runtime_Error_Code := 1;
    L_Runtime_Error_Text := 'Gas valve not closed';
END_IF;

// GAS: ventilation must not be forced fully off by the IO layer.
IF (NOT L_Runtime_Error) AND (GVL_SAFETY_SHUTDOWN.G_Safety_Mode = GAS) THEN
    IF (GVL_IO.AO_Supply_Fans[1] = 0) AND (GVL_IO.AO_Exhaust_Fans[1] = 0) THEN
        L_Runtime_Error := TRUE;
        L_Runtime_Error_Code := 3;
        L_Runtime_Error_Text := 'Gas ventilation inactive';
    END_IF;
END_IF;

// FIRE: all exhaust fans should be commanded above zero in smoke exhaust mode.
IF (NOT L_Runtime_Error) AND (GVL_SAFETY_SHUTDOWN.G_Safety_Mode = FIRE) THEN
    FOR L_i := 1 TO GVL_CONSTANTS.C_MAX_EXHAUST_FANS DO
        IF GVL_IO.AO_Exhaust_Fans[L_i] = 0 THEN
            L_Runtime_Error := TRUE;
            L_Runtime_Error_Code := 2;
            L_Runtime_Error_Text := 'Smoke exhaust not active';
        END_IF;
    END_FOR;
END_IF;

// FIRE: supply fans should be off in smoke exhaust mode.
IF (NOT L_Runtime_Error) AND (GVL_SAFETY_SHUTDOWN.G_Safety_Mode = FIRE) THEN
    FOR L_i := 1 TO GVL_CONSTANTS.C_MAX_SUPPLY_FANS DO
        IF GVL_IO.AO_Supply_Fans[L_i] <> 0 THEN
            L_Runtime_Error := TRUE;
            L_Runtime_Error_Code := 4;
            L_Runtime_Error_Text := 'Supply fan active in fire';
        END_IF;
    END_FOR;
END_IF;

// WATER_LEAK: valve close commands must reach physical outputs.
IF (NOT L_Runtime_Error) AND (GVL_SAFETY_SHUTDOWN.G_Safety_Mode = WATER_LEAK) THEN
    IF GVL_COMMAND_SHADOW.G_Close_Valve_35 AND (NOT GVL_IO.DO_Water_Valve_35_Close) THEN
        L_Runtime_Error := TRUE;
        L_Runtime_Error_Code := 5;
        L_Runtime_Error_Text := 'Water valve 35 not closed';
    ELSIF GVL_COMMAND_SHADOW.G_Close_Valve_36 AND (NOT GVL_IO.DO_Water_Valve_36_Close) THEN
        L_Runtime_Error := TRUE;
        L_Runtime_Error_Code := 6;
        L_Runtime_Error_Text := 'Water valve 36 not closed';
    END_IF;
END_IF;

// FREEZE: when freeze-risk is active, heating circulation should not be fully dead.
IF (NOT L_Runtime_Error) AND GVL_STATE.G_Safety_Freeze_Risk THEN
    FOR L_i := 1 TO GVL_CONSTANTS.C_MAX_MANIFOLDS DO
        IF GVL_IO.DO_Manifold_Pumps[L_i] THEN
            L_Any_Manifold_Pump_On := TRUE;
        END_IF;
    END_FOR;

    IF (NOT L_Any_Manifold_Pump_On) AND (NOT GVL_IO.DO_Backup_Circulation_Pump) THEN
        L_Runtime_Error := TRUE;
        L_Runtime_Error_Code := 7;
        L_Runtime_Error_Text := 'Freeze circulation inactive';
    END_IF;
END_IF;

// GAS+FREEZE: electric backup may be used for anti-freeze, but DHW heating must remain off.
IF (NOT L_Runtime_Error) AND GVL_STATE.G_Safety_Freeze_Risk AND GVL_COMMAND_SHADOW.G_Heating_Gas_Safety_Stop THEN
    IF GVL_IO.DO_DHW_Heating_Pump THEN
        L_Runtime_Error := TRUE;
        L_Runtime_Error_Code := 8;
        L_Runtime_Error_Text := 'DHW heating active during gas freeze';
    END_IF;
END_IF;

// Apply result
IF L_Runtime_Error THEN
    GVL_COMMAND_VERIFY.Runtime_Sanity_OK := FALSE;
    GVL_COMMAND_VERIFY.Runtime_Last_Error_Code := L_Runtime_Error_Code;
    GVL_COMMAND_VERIFY.Runtime_Last_Error_Text := L_Runtime_Error_Text;
    GVL_COMMAND_VERIFY.Runtime_Last_Error_Time_MS := L_Now_MS;

    IF NOT L_Prev_Runtime_Error THEN
        GVL_COMMAND_VERIFY.Runtime_Sanity_Error_Count := GVL_COMMAND_VERIFY.Runtime_Sanity_Error_Count + 1;
        fbLog(
            VI_Event_Type := 1001,
            VI_Timestamp := L_Now_MS,
            VI_Param1 := L_Runtime_Error_Code,
            VI_Param2 := GVL_COMMAND_VERIFY.Runtime_Sanity_Error_Count
        );
    END_IF;
ELSE
    GVL_COMMAND_VERIFY.Runtime_Sanity_OK := TRUE;
END_IF;

L_Prev_Runtime_Error := L_Runtime_Error;

END_PROGRAM

(* ---- PRG_Config_Validation.st ---- *)
PROGRAM PRG_Config_Validation
VAR
    fbConfigSimulation : FB_Config_Simulation;

    L_i : INT;
    L_Zone : INT;
    L_Sensor : INT;
    L_Manifold : INT;
    L_Map_Index : INT;
    L_Config_Error : BOOL;
END_VAR

// ======================================================
// CENTRAL CONFIGURATION VALIDATION
// ======================================================
// Diagnostic-only layer.
//
// This PRG may set validation/configuration status flags and text,
// but must not directly mutate aggregated diagnostics fields.
// Aggregated diagnostics ownership is centralized in:
//
//   FB_System_Health_Orchestrator
//
// This PRG also must not write command/shadow/output structures.
// ======================================================

L_Config_Error := FALSE;

// ======================================================
// ACTIVE SIZE CONFIGURATION
// ======================================================
IF (GVL_SYSTEM_SIZE_CONFIG.G_Active_Heating_Circuits < 1) OR
   (GVL_SYSTEM_SIZE_CONFIG.G_Active_Heating_Circuits > GVL_CONSTANTS.C_MAX_HEATING_CIRCUITS) THEN
    L_Config_Error := TRUE;
END_IF;

IF (GVL_SYSTEM_SIZE_CONFIG.G_Active_Water_Zones < 1) OR
   (GVL_SYSTEM_SIZE_CONFIG.G_Active_Water_Zones > GVL_CONSTANTS.C_MAX_WATER_ZONES) THEN
    L_Config_Error := TRUE;
END_IF;

IF (GVL_SYSTEM_SIZE_CONFIG.G_Active_Light_Zones < 1) OR
   (GVL_SYSTEM_SIZE_CONFIG.G_Active_Light_Zones > GVL_CONSTANTS.C_MAX_LIGHT_ZONES) THEN
    L_Config_Error := TRUE;
END_IF;

IF (GVL_SYSTEM_SIZE_CONFIG.G_Active_Blinds < 0) OR
   (GVL_SYSTEM_SIZE_CONFIG.G_Active_Blinds > GVL_CONSTANTS.C_MAX_BLINDS) THEN
    L_Config_Error := TRUE;
END_IF;

IF (GVL_SYSTEM_SIZE_CONFIG.G_Active_Sockets < 0) OR
   (GVL_SYSTEM_SIZE_CONFIG.G_Active_Sockets > GVL_CONSTANTS.C_MAX_SOCKETS) THEN
    L_Config_Error := TRUE;
END_IF;

// ======================================================
// HEATING CIRCUIT CONFIGURATION
// ======================================================
FOR L_i := 1 TO GVL_CONSTANTS.C_MAX_HEATING_CIRCUITS DO
    L_Zone := BYTE_TO_INT(GVL_CONFIG.G_HMI_FloorHeating_Configs[L_i].zone);
    L_Sensor := BYTE_TO_INT(GVL_CONFIG.G_HMI_FloorHeating_Configs[L_i].sensor_id);
    L_Manifold := BYTE_TO_INT(GVL_CONFIG.G_HMI_FloorHeating_Configs[L_i].manifold_id);

    IF (L_Zone < 1) OR (L_Zone > GVL_CONSTANTS.C_MAX_ZONES) THEN
        L_Config_Error := TRUE;
    END_IF;

    IF (L_Sensor < 1) OR (L_Sensor > GVL_CONSTANTS.C_MAX_ZONES) THEN
        L_Config_Error := TRUE;
    END_IF;

    IF (L_Manifold < 1) OR (L_Manifold > GVL_CONSTANTS.C_MAX_MANIFOLDS) THEN
        L_Config_Error := TRUE;
    END_IF;

    IF GVL_CONFIG.G_HMI_FloorHeating_Configs[L_i].min_temp > GVL_CONFIG.G_HMI_FloorHeating_Configs[L_i].max_temp THEN
        L_Config_Error := TRUE;
    END_IF;
END_FOR;

IF (GVL_CONFIG.G_Max_Active_Manifolds < 1) OR
   (GVL_CONFIG.G_Max_Active_Manifolds > GVL_CONSTANTS.C_MAX_MANIFOLDS) THEN
    L_Config_Error := TRUE;
END_IF;

IF GVL_CONFIG.G_Max_Thermal_Budget <= 0.0 THEN
    L_Config_Error := TRUE;
END_IF;

IF GVL_CONFIG.G_Policy_Min_Hold_MS < 10000 THEN
    L_Config_Error := TRUE;
END_IF;

// ======================================================
// ACCESS / TIMING CONFIGURATION
// ======================================================
IF (GVL_CONFIG.G_Access_Pulse_MS < 100) OR (GVL_CONFIG.G_Access_Pulse_MS > 5000) THEN
    L_Config_Error := TRUE;
END_IF;

// ======================================================
// MAP CONFIGURATION
// ======================================================
FOR L_i := 1 TO GVL_CONSTANTS.C_MAX_DOOR_SENSORS DO
    L_Map_Index := GVL_CONFIG.G_Door_Map[L_i];
    IF (L_Map_Index < 1) OR (L_Map_Index > GVL_CONSTANTS.C_MAX_SECURITY_SENSORS) THEN
        L_Config_Error := TRUE;
    END_IF;
END_FOR;

FOR L_i := 1 TO GVL_CONSTANTS.C_MAX_ZONES DO
    L_Map_Index := GVL_CONFIG.G_Window_Map[L_i];
    IF L_Map_Index <> 0 THEN
        IF (L_Map_Index < 1) OR (L_Map_Index > (GVL_CONSTANTS.C_MAX_SECURITY_SENSORS * 2)) THEN
            L_Config_Error := TRUE;
        END_IF;
    END_IF;
END_FOR;

FOR L_i := 1 TO GVL_CONSTANTS.C_MAX_HEATING_CIRCUITS DO
    IF (GVL_CONFIG.G_FloorTemp_Map[L_i] < 1) OR (GVL_CONFIG.G_FloorTemp_Map[L_i] > GVL_CONSTANTS.C_MAX_ZONES) THEN
        L_Config_Error := TRUE;
    END_IF;
END_FOR;

FOR L_i := 1 TO GVL_CONSTANTS.C_MAX_ZONES DO
    IF (GVL_CONFIG.G_RoomTemp_Map[L_i] < 1) OR (GVL_CONFIG.G_RoomTemp_Map[L_i] > GVL_CONSTANTS.C_MAX_ZONES) THEN
        L_Config_Error := TRUE;
    END_IF;
END_FOR;

// ======================================================
// HARDWARE SERVICE / RETRY CONFIGURATION
// ======================================================
IF GVL_CONFIG.G_Freeze_Hardware_Retry_Count < 0 THEN
    L_Config_Error := TRUE;
END_IF;

IF GVL_CONFIG.G_Freeze_Hardware_Retry_Delay_MS < 1000 THEN
    L_Config_Error := TRUE;
END_IF;

IF GVL_CONFIG.G_Pump_Exercise_Enabled THEN
    IF GVL_CONFIG.G_Pump_Exercise_Interval_MS < GVL_CONSTANTS.C_MS_IN_MINUTE THEN
        L_Config_Error := TRUE;
    END_IF;
    IF GVL_CONFIG.G_Pump_Exercise_Duration_MS < 1000 THEN
        L_Config_Error := TRUE;
    END_IF;
END_IF;

IF GVL_CONFIG.G_Water_Valve_Exercise_Enabled THEN
    IF GVL_CONFIG.G_Water_Valve_Exercise_Interval_MS < GVL_CONSTANTS.C_MS_IN_MINUTE THEN
        L_Config_Error := TRUE;
    END_IF;
    IF GVL_CONFIG.G_Water_Valve_Exercise_Duration_MS < 1000 THEN
        L_Config_Error := TRUE;
    END_IF;
END_IF;

IF GVL_CONFIG.G_Water_Valve_Close_Retry_Count < 0 THEN
    L_Config_Error := TRUE;
END_IF;

IF GVL_CONFIG.G_Water_Valve_Close_Retry_Delay_MS < 1000 THEN
    L_Config_Error := TRUE;
END_IF;

// ======================================================
// OPENTHERM / MODBUS RTU CONFIGURATION
// ======================================================
IF GVL_CONFIG.G_OpenTherm_Enabled THEN

    IF GVL_CONFIG.G_OpenTherm_Heartbeat_Timeout_MS < 1000 THEN
        L_Config_Error := TRUE;
    END_IF;

    IF GVL_CONFIG.G_OpenTherm_Command_Ack_Timeout_MS < 500 THEN
        L_Config_Error := TRUE;
    END_IF;

    IF GVL_CONFIG.G_Modbus_RTU_Baudrate < 1200 THEN
        L_Config_Error := TRUE;
    END_IF;

    IF (GVL_CONFIG.G_Modbus_RTU_Parity > 2) THEN
        L_Config_Error := TRUE;
    END_IF;

    IF (GVL_CONFIG.G_Modbus_RTU_Stop_Bits < 1) OR
       (GVL_CONFIG.G_Modbus_RTU_Stop_Bits > 2) THEN
        L_Config_Error := TRUE;
    END_IF;

    IF (GVL_CONFIG.G_Modbus_RTU_Data_Bits < 7) OR
       (GVL_CONFIG.G_Modbus_RTU_Data_Bits > 8) THEN
        L_Config_Error := TRUE;
    END_IF;

    IF GVL_CONFIG.G_Modbus_RTU_Slave_ID = 0 THEN
        L_Config_Error := TRUE;
    END_IF;

    IF GVL_CONFIG.G_Modbus_RTU_Poll_Interval_MS < 50 THEN
        L_Config_Error := TRUE;
    END_IF;

    IF GVL_CONFIG.G_Modbus_RTU_Request_Timeout_MS < 50 THEN
        L_Config_Error := TRUE;
    END_IF;

    IF GVL_CONFIG.G_Modbus_RTU_Retry_Count < 0 THEN
        L_Config_Error := TRUE;
    END_IF;

    FOR L_i := 1 TO GVL_CONSTANTS.C_MAX_BOILERS DO
        IF GVL_CONFIG.G_OpenTherm_Register_Map[L_i].Cmd_Enable_Offset = GVL_CONFIG.G_OpenTherm_Register_Map[L_i].Status_Word_Offset THEN
            L_Config_Error := TRUE;
        END_IF;

        IF GVL_CONFIG.G_OpenTherm_Register_Map[L_i].Cmd_Setpoint_x10_Offset = GVL_CONFIG.G_OpenTherm_Register_Map[L_i].Status_Word_Offset THEN
            L_Config_Error := TRUE;
        END_IF;
    END_FOR;
END_IF;

// ======================================================
// SENSOR COUNT SANITY
// ======================================================
IF GVL_CONSTANTS.C_MAX_METHANE_SENSORS < 2 THEN
    L_Config_Error := TRUE;
END_IF;

IF GVL_CONSTANTS.C_MAX_SMOKE_SENSORS < 6 THEN
    L_Config_Error := TRUE;
END_IF;

IF GVL_CONSTANTS.C_MAX_CO_SENSORS < 8 THEN
    L_Config_Error := TRUE;
END_IF;

IF GVL_CONSTANTS.C_MAX_FLOOD_SENSORS < 9 THEN
    L_Config_Error := TRUE;
END_IF;

// ======================================================
// CONFIG SIMULATION / COMMISSIONING VALIDATION
// ======================================================
fbConfigSimulation(
    VI_Enable := TRUE,
    VI_Request := GVL_CONFIG_SIMULATION.G_Simulation_Request,
    VI_Confirm := GVL_CONFIG_SIMULATION.G_Simulation_Confirm
);

IF fbConfigSimulation.VO_Executed AND NOT fbConfigSimulation.VO_Result_OK THEN
    L_Config_Error := TRUE;
END_IF;

// ======================================================
// STORE FLAGS
// ======================================================
GVL_CONFIG_VALIDATION.G_Config_Valid := NOT L_Config_Error;
GVL_CONFIG_VALIDATION.G_Config_Critical_Error := L_Config_Error;
GVL_CONFIG_VALIDATION.G_Config_Last_Update_MS := GVL_STATUS.G_System_Time_MS;

IF L_Config_Error THEN
    GVL_CONFIG_VALIDATION.G_Config_Last_Error_Text := 'CONFIG VALIDATION ERROR';
    GVL_STATUS.G_System_Mode_Text := 'CONFIG ERROR';
ELSE
    GVL_CONFIG_VALIDATION.G_Config_Last_Error_Text := '';
END_IF;

END_PROGRAM

(* ---- PRG_Control_Temporal_Coherence_Governor.st ---- *)
PROGRAM PRG_Control_Temporal_Coherence_Governor
VAR
    L_Now_MS : UDINT;
    L_Control_Valid : BOOL := TRUE;
    L_Error_Code : UDINT := 0;
    L_Error_Text : STRING(160) := '';
END_VAR

L_Now_MS := GVL_STATUS.G_System_Time_MS;
L_Control_Valid := TRUE;
L_Error_Code := 0;
L_Error_Text := '';

// Fail-safe defaults.
GVL_CONTROL_TIMING_FABRIC.Control_Temporal_Coherence_Valid := FALSE;
GVL_CONTROL_TIMING_FABRIC.Control_Temporal_Coherence_Granted := FALSE;
GVL_CONTROL_TIMING_FABRIC.Control_Temporal_Coherence_Quarantine_Active := TRUE;

GVL_CONTROL_TIMING_FABRIC.Loop_Sampling_Coherent := FALSE;
GVL_CONTROL_TIMING_FABRIC.Feedback_Freshness_Valid := FALSE;
GVL_CONTROL_TIMING_FABRIC.PID_Phase_Alignment_Valid := FALSE;
GVL_CONTROL_TIMING_FABRIC.Cross_Loop_Temporal_Stable := FALSE;
GVL_CONTROL_TIMING_FABRIC.Multi_Rate_Causality_Coherent := FALSE;

// Global authority synchronization required.
IF NOT GVL_GLOBAL_AUTHORITY_SYNC.Global_Authority_Sync_Granted THEN
    L_Control_Valid := FALSE;
    L_Error_Code := 35000;
    L_Error_Text := 'Global authority synchronization not granted';
END_IF;

// Temporal aliasing detectors.
IF GVL_CONTROL_TIMING_FABRIC.PID_Phase_Skew_Detected THEN
    L_Control_Valid := FALSE;
    L_Error_Code := 35001;
    L_Error_Text := 'PID phase skew detected';
END_IF;

IF GVL_CONTROL_TIMING_FABRIC.Sampling_Window_Divergence_Detected THEN
    L_Control_Valid := FALSE;
    L_Error_Code := 35002;
    L_Error_Text := 'Sampling window divergence detected';
END_IF;

IF GVL_CONTROL_TIMING_FABRIC.Feedback_Freshness_Aliasing_Detected THEN
    L_Control_Valid := FALSE;
    L_Error_Code := 35003;
    L_Error_Text := 'Feedback freshness aliasing detected';
END_IF;

IF GVL_CONTROL_TIMING_FABRIC.Cross_Loop_Stabilization_Lag_Detected THEN
    L_Control_Valid := FALSE;
    L_Error_Code := 35004;
    L_Error_Text := 'Cross-loop stabilization lag detected';
END_IF;

IF GVL_CONTROL_TIMING_FABRIC.Multi_Rate_Oscillation_Risk_Detected THEN
    L_Control_Valid := FALSE;
    L_Error_Code := 35005;
    L_Error_Text := 'Multi-rate oscillation risk detected';
END_IF;

IF GVL_CONTROL_TIMING_FABRIC.Distributed_Control_Ringing_Detected THEN
    L_Control_Valid := FALSE;
    L_Error_Code := 35006;
    L_Error_Text := 'Distributed control ringing detected';
END_IF;

// Deterministic control timing validation.
IF L_Control_Valid
AND NOT GVL_CONTROL_TIMING_FABRIC.Control_Snapshot_Epoch_Coherent THEN
    L_Control_Valid := FALSE;
    L_Error_Code := 35010;
    L_Error_Text := 'Control snapshot epoch coherence invalid';
END_IF;

IF L_Control_Valid
AND NOT GVL_CONTROL_TIMING_FABRIC.Feedback_Window_Stable THEN
    L_Control_Valid := FALSE;
    L_Error_Code := 35011;
    L_Error_Text := 'Feedback window unstable';
END_IF;

IF L_Control_Valid
AND NOT GVL_CONTROL_TIMING_FABRIC.Loop_Execution_Phase_Stable THEN
    L_Control_Valid := FALSE;
    L_Error_Code := 35012;
    L_Error_Text := 'Loop execution phase unstable';
END_IF;

IF L_Control_Valid
AND NOT GVL_CONTROL_TIMING_FABRIC.Temporal_Observation_Aligned THEN
    L_Control_Valid := FALSE;
    L_Error_Code := 35013;
    L_Error_Text := 'Temporal observation alignment invalid';
END_IF;

IF L_Control_Valid THEN
    GVL_CONTROL_TIMING_FABRIC.Control_Temporal_Coherence_Valid := TRUE;
    GVL_CONTROL_TIMING_FABRIC.Control_Temporal_Coherence_Granted := TRUE;
    GVL_CONTROL_TIMING_FABRIC.Control_Temporal_Coherence_Quarantine_Active := FALSE;

    GVL_CONTROL_TIMING_FABRIC.Loop_Sampling_Coherent := TRUE;
    GVL_CONTROL_TIMING_FABRIC.Feedback_Freshness_Valid := TRUE;
    GVL_CONTROL_TIMING_FABRIC.PID_Phase_Alignment_Valid := TRUE;
    GVL_CONTROL_TIMING_FABRIC.Cross_Loop_Temporal_Stable := TRUE;
    GVL_CONTROL_TIMING_FABRIC.Multi_Rate_Causality_Coherent := TRUE;

    GVL_CONTROL_TIMING_FABRIC.Control_Timing_Epoch :=
        GVL_GLOBAL_AUTHORITY_SYNC.Global_Authority_Epoch;

    GVL_CONTROL_TIMING_FABRIC.Control_Timing_Epoch_Coherent := TRUE;

    GVL_CONTROL_TIMING_FABRIC.Control_Timing_Last_Update_MS := L_Now_MS;
    GVL_CONTROL_TIMING_FABRIC.Control_Timing_Lease_Expired := FALSE;

    GVL_CONTROL_TIMING_FABRIC.Control_Timing_Last_Error_Code := 0;
    GVL_CONTROL_TIMING_FABRIC.Control_Timing_Last_Error_Text := '';
ELSE
    GVL_CONTROL_TIMING_FABRIC.Control_Temporal_Coherence_Valid := FALSE;
    GVL_CONTROL_TIMING_FABRIC.Control_Temporal_Coherence_Granted := FALSE;
    GVL_CONTROL_TIMING_FABRIC.Control_Temporal_Coherence_Quarantine_Active := TRUE;

    GVL_CONTROL_TIMING_FABRIC.Control_Timing_Lease_Expired := TRUE;

    GVL_CONTROL_TIMING_FABRIC.Control_Timing_Last_Error_Code :=
        L_Error_Code;

    GVL_CONTROL_TIMING_FABRIC.Control_Timing_Last_Error_Text :=
        L_Error_Text;

    GVL_CONTROL_TIMING_FABRIC.Control_Timing_Invalidation_Count :=
        GVL_CONTROL_TIMING_FABRIC.Control_Timing_Invalidation_Count + 1;
END_IF;

END_PROGRAM

(* ---- PRG_Controlled_Capability_Shedding_Governor.st ---- *)
PROGRAM PRG_Controlled_Capability_Shedding_Governor
// CONTROLLED CAPABILITY SHEDDING
// DETERMINISTIC / TIER-AWARE / NON-INVASIVE

IF GVL_RUNTIME_BUDGET_ENFORCEMENT.Runtime_Budget_Pressure_Observed THEN
    GVL_FABRIC_LIFECYCLE_REGISTRY.Controlled_Capability_Shedding_Allowed := TRUE;
    GVL_FABRIC_LIFECYCLE_REGISTRY.Runtime_Adaptive_Mode := REDUCED_ANALYTICS_MODE;
END_IF;

IF GVL_SURVIVABILITY_INTELLIGENCE_FABRIC.Chronic_Degradation_Risk_Increasing THEN
    GVL_FABRIC_LIFECYCLE_REGISTRY.Runtime_Adaptive_Mode := SURVIVABILITY_MODE;
    GVL_FABRIC_LIFECYCLE_REGISTRY.NonEssential_Analytics_Shedding_Recommended := TRUE;
    GVL_FABRIC_LIFECYCLE_REGISTRY.Diagnostics_Degradation_Recommended := TRUE;
END_IF;

IF GVL_RUNTIME_BUDGET_ENFORCEMENT.Verification_Induced_Runtime_Risk THEN
    GVL_FABRIC_LIFECYCLE_REGISTRY.Extended_Observability_Shedding_Recommended := TRUE;
    GVL_FABRIC_LIFECYCLE_REGISTRY.Simulation_Suspension_Recommended := TRUE;
END_IF;

IF GVL_RUNTIME_BUDGET_ENFORCEMENT.Runtime_Stability_Budget_At_Risk THEN
    GVL_FABRIC_LIFECYCLE_REGISTRY.Analytics_Fabric_State := FABRIC_DEGRADED;
    GVL_FABRIC_LIFECYCLE_REGISTRY.Observability_Fabric_State := FABRIC_PASSIVE;
END_IF;

// Critical fabrics remain protected.
GVL_FABRIC_LIFECYCLE_REGISTRY.Safety_Fabric_State := FABRIC_ACTIVE;
GVL_FABRIC_LIFECYCLE_REGISTRY.Authority_Fabric_State := FABRIC_ACTIVE;
GVL_FABRIC_LIFECYCLE_REGISTRY.Physical_Reality_Fabric_State := FABRIC_ACTIVE;

IF NOT GVL_RUNTIME_BUDGET_ENFORCEMENT.Runtime_Budget_Pressure_Observed THEN
    GVL_FABRIC_LIFECYCLE_REGISTRY.Gradual_Reactivation_Allowed := TRUE;
END_IF;

END_PROGRAM

(* ---- PRG_Debug_View.st ---- *)
PROGRAM PRG_Debug_View
VAR
    L_i : INT;
    L_MaxWeight : REAL;
    L_MinWeight : REAL;
    L_Weight : REAL;
    L_Index : INT;
END_VAR

GVL_DEBUG_VIEW.D_Current_Time_MS := GVL_TIME_SERVICE.G_Now_MS;

GVL_DEBUG_VIEW.D_Safety_Mode := GVL_SAFETY_SHUTDOWN.G_Safety_Mode;
GVL_DEBUG_VIEW.D_Safety_Active := (GVL_SAFETY_SHUTDOWN.G_Safety_Mode <> NORMAL);
GVL_DEBUG_VIEW.D_Recovery_Phase := GVL_SAFETY_RECOVERY.G_Recovery_Phase;
GVL_DEBUG_VIEW.D_Recovery_Active := GVL_SAFETY_RECOVERY.G_Recovery_Active;

GVL_DEBUG_VIEW.D_Current_Scenario := GVL_INTENT_BEHAVIOR.I_Selected_Scenario_Text;
GVL_DEBUG_VIEW.D_Behavior_Reason := GVL_INTENT_BEHAVIOR.I_Reason_Text;

GVL_DEBUG_VIEW.D_Score_Night := GVL_INTENT_BEHAVIOR.I_Score_Night;
GVL_DEBUG_VIEW.D_Score_Preheat := GVL_INTENT_BEHAVIOR.I_Score_Preheat;
GVL_DEBUG_VIEW.D_Score_VentBoost := GVL_INTENT_BEHAVIOR.I_Score_Vent_Boost;
GVL_DEBUG_VIEW.D_Score_AccessSecure := GVL_INTENT_BEHAVIOR.I_Score_Access_Secure;

GVL_DEBUG_VIEW.D_Intent_Night := GVL_INTENT_BEHAVIOR.I_Request_Night_Mode;
GVL_DEBUG_VIEW.D_Intent_Comfort := GVL_INTENT_BEHAVIOR.I_Request_Comfort_Mode;
GVL_DEBUG_VIEW.D_Intent_VentBoost := GVL_INTENT_BEHAVIOR.I_Request_Ventilation_Boost;
GVL_DEBUG_VIEW.D_Intent_AccessSecure := GVL_INTENT_BEHAVIOR.I_Request_Access_Secure_Mode;

GVL_DEBUG_VIEW.D_Heating_Block := GVL_COMMAND_SHADOW.G_Heating_Block;
GVL_DEBUG_VIEW.D_Vent_Stop := GVL_COMMAND_SHADOW.G_Vent_Stop;
GVL_DEBUG_VIEW.D_Water_Block := GVL_COMMAND_SHADOW.G_Water_Block;
GVL_DEBUG_VIEW.D_Access_Open_Active := GVL_COMMAND_SHADOW.G_Gate_Open OR GVL_COMMAND_SHADOW.G_Wicket_Open;

GVL_DEBUG_VIEW.D_Global_Reason := GVL_EXPLAINABILITY.G_Last_Global_Reason_Text;
GVL_DEBUG_VIEW.D_Behavior_Why_Active := GVL_EXPLAINABILITY.G_Behavior_Why_Active;
GVL_DEBUG_VIEW.D_Heating_Why_Blocked := GVL_EXPLAINABILITY.G_Heating_Why_Blocked;
GVL_DEBUG_VIEW.D_Vent_Why_Stopped := GVL_EXPLAINABILITY.G_Vent_Why_Stopped;
GVL_DEBUG_VIEW.D_Water_Why_Closed := GVL_EXPLAINABILITY.G_Water_Why_Closed;
GVL_DEBUG_VIEW.D_Access_Why_Opened := GVL_EXPLAINABILITY.G_Access_Why_Opened;

// SENSOR QUALITY → HMI
GVL_DEBUG_VIEW.D_Input_Source_Valid := GVL_INPUT.IN_Source_Valid;
GVL_DEBUG_VIEW.D_Input_Degraded := GVL_INPUT.IN_Input_Degraded;
GVL_DEBUG_VIEW.D_Sensor_Fault := GVL_INPUT.IN_Sensor_Fault;
GVL_DEBUG_VIEW.D_Validation_Failed := GVL_INPUT.IN_Validation_Failed;
GVL_DEBUG_VIEW.D_Anomaly_Detected := GVL_INPUT.IN_Anomaly_Detected;
GVL_DEBUG_VIEW.D_Validation_Reason := GVL_INPUT.IN_Validation_Reason;
GVL_DEBUG_VIEW.D_Anomaly_Reason := GVL_INPUT.IN_Anomaly_Reason;
GVL_DEBUG_VIEW.D_Last_Invalid_Zone := GVL_INPUT.IN_Last_Invalid_Zone;
GVL_DEBUG_VIEW.D_Min_Zone_Confidence := GVL_INPUT.IN_Min_Zone_Confidence;
GVL_DEBUG_VIEW.D_Worst_Zone := GVL_INPUT.IN_Worst_Zone;

GVL_DEBUG_VIEW.D_Adapt_Profile := GVL_BEHAVIOR_ADAPT.G_Adapt_Profile;

IF GVL_BEHAVIOR_ADAPT.G_Adapt_Profile = ADAPT_PROFILE_STABLE THEN
    GVL_DEBUG_VIEW.D_Adapt_Profile_Text := 'STABLE';
ELSIF GVL_BEHAVIOR_ADAPT.G_Adapt_Profile = ADAPT_PROFILE_BALANCED THEN
    GVL_DEBUG_VIEW.D_Adapt_Profile_Text := 'BALANCED';
ELSE
    GVL_DEBUG_VIEW.D_Adapt_Profile_Text := 'AGGRESSIVE';
END_IF;

L_MaxWeight := 0.0;
L_MinWeight := 9999.0;
GVL_DEBUG_VIEW.D_Main_VentBoost_Zone := 0;

FOR L_i := 1 TO GVL_CONSTANTS.C_MAX_ZONES DO
    L_Weight := GVL_BEHAVIOR_ADAPT.G_VentBoost_Zone_Adapt[L_i].Zone_Weight;
    IF L_Weight > L_MaxWeight THEN
        L_MaxWeight := L_Weight;
        GVL_DEBUG_VIEW.D_Main_VentBoost_Zone := L_i;
        GVL_DEBUG_VIEW.D_Main_VentBoost_Zone_Weight := L_Weight;
        GVL_DEBUG_VIEW.D_Main_VentBoost_Zone_Confidence :=
            GVL_BEHAVIOR_ADAPT.G_VentBoost_Zone_Adapt[L_i].Confidence;
    END_IF;
    IF L_Weight < L_MinWeight THEN
        L_MinWeight := L_Weight;
    END_IF;
END_FOR;

GVL_DEBUG_VIEW.D_Max_VentBoost_Zone_Weight := L_MaxWeight;
GVL_DEBUG_VIEW.D_Min_VentBoost_Zone_Weight := L_MinWeight;

L_Index := GVL_TRACE.G_Trace_Write_Index - 1;
IF L_Index < 1 THEN
    L_Index := 200;
END_IF;

GVL_DEBUG_VIEW.D_Last_Trace_Text := GVL_TRACE.G_Trace_Buffer[L_Index].Text;
GVL_DEBUG_VIEW.D_Last_Trace_Time_MS := GVL_TRACE.G_Trace_Buffer[L_Index].Timestamp_MS;
GVL_DEBUG_VIEW.D_Last_Trace_Reason := GVL_TRACE.G_Trace_Buffer[L_Index].Reason_Code;

END_PROGRAM

(* ---- PRG_Distributed_Commit_Governor.st ---- *)
PROGRAM PRG_Distributed_Commit_Governor
VAR
    L_Now_MS : UDINT;
    L_Delta_MS : UDINT;
    L_Commit_Valid : BOOL := TRUE;
    L_Error_Code : UDINT := 0;
    L_Error_Text : STRING(160) := '';
    L_Peer_Session_Active : BOOL := FALSE;

    L_Publication_Authority_Allowed : BOOL;
END_VAR

L_Now_MS := GVL_STATUS.G_System_Time_MS;
L_Commit_Valid := TRUE;
L_Error_Code := 0;
L_Error_Text := '';

GVL_DISTRIBUTED_COMMIT.Peer_Commit_Ack_Expired := FALSE;
GVL_DISTRIBUTED_COMMIT.Peer_Commit_Mismatch := FALSE;
GVL_DISTRIBUTED_COMMIT.Peer_Commit_Replay_Detected := FALSE;
GVL_DISTRIBUTED_COMMIT.Peer_Commit_Missing := FALSE;
GVL_DISTRIBUTED_COMMIT.Commit_Lease_Expired := FALSE;

// Finalized publication/convergence authority.
L_Publication_Authority_Allowed :=
    GVL_Distributed_Execution_Gates.G_Runtime_Valid
    AND GVL_Distributed_Execution_Gates.G_Can_Replicate
    AND GVL_Distributed_Execution_Gates.G_Can_Own_Projection
    AND GVL_CONVERGENCE.Convergence_Lease_OK
    AND GVL_CONVERGENCE.Convergence_Release_Allowed
    AND GVL_RECOVERY_GOVERNANCE.Recovery_Governance_Valid
    AND NOT GVL_RECOVERY_GOVERNANCE.Recovery_Quarantine_Active;

GVL_DISTRIBUTED_COMMIT.Local_Publication_Commit_Epoch := GVL_DISTRIBUTED_SNAPSHOT.Distributed_Snapshot_Epoch;
GVL_DISTRIBUTED_COMMIT.Local_Prepare_Epoch := GVL_DISTRIBUTED_SNAPSHOT.Distributed_Snapshot_Epoch;

IF NOT L_Publication_Authority_Allowed THEN

    L_Commit_Valid := FALSE;

    L_Error_Code := 14999;
    L_Error_Text :=
        'Distributed publication authority restricted';

END_IF;

IF L_Commit_Valid THEN

    IF GVL_DISTRIBUTED_SNAPSHOT.Distributed_Publication_Reconciled
    AND GVL_DISTRIBUTED_SNAPSHOT.Distributed_Publication_Freeze_Valid
    AND GVL_DISTRIBUTED_SNAPSHOT.Distributed_Snapshot_Consistent
    THEN
        GVL_DISTRIBUTED_COMMIT.Publication_Prepare_Active := TRUE;
        GVL_DISTRIBUTED_COMMIT.Publication_Prepare_Valid := TRUE;
    ELSE
        GVL_DISTRIBUTED_COMMIT.Publication_Prepare_Active := FALSE;
        GVL_DISTRIBUTED_COMMIT.Publication_Prepare_Valid := FALSE;

        L_Commit_Valid := FALSE;
        L_Error_Code := 15000;
        L_Error_Text := 'Distributed immutable publication prepare invalid';
    END_IF;

END_IF;

IF GVL_DISTRIBUTED_COMMIT.Peer_Publication_Commit_Epoch > 0 THEN
    L_Peer_Session_Active := TRUE;
END_IF;

IF GVL_DISTRIBUTED_COMMIT.Peer_Prepare_Epoch > 0 THEN
    L_Peer_Session_Active := TRUE;
END_IF;

IF GVL_DISTRIBUTED_COMMIT.Peer_Commit_Ack_Valid THEN
    L_Peer_Session_Active := TRUE;
END_IF;

IF L_Commit_Valid AND L_Peer_Session_Active THEN
    L_Delta_MS := L_Now_MS - GVL_DISTRIBUTED_COMMIT.Peer_Commit_Last_Refresh_MS;

    IF GVL_DISTRIBUTED_COMMIT.Commit_Lease_Active THEN
        IF L_Delta_MS > GVL_DISTRIBUTED_COMMIT.Commit_Timeout_MS THEN
            GVL_DISTRIBUTED_COMMIT.Commit_Lease_Expired := TRUE;

            L_Commit_Valid := FALSE;
            L_Error_Code := 15001;
            L_Error_Text := 'Distributed commit lease expired';
        END_IF;
    END_IF;
END_IF;

IF L_Commit_Valid AND L_Peer_Session_Active THEN
    IF NOT GVL_DISTRIBUTED_COMMIT.Peer_Commit_Ack_Valid THEN
        GVL_DISTRIBUTED_COMMIT.Peer_Commit_Missing := TRUE;

        L_Commit_Valid := FALSE;
        L_Error_Code := 15002;
        L_Error_Text := 'Peer commit acknowledgement missing';
    END_IF;
END_IF;

IF L_Commit_Valid AND L_Peer_Session_Active THEN
    IF GVL_DISTRIBUTED_COMMIT.Peer_Publication_Commit_Epoch < GVL_DISTRIBUTED_COMMIT.Local_Publication_Commit_Epoch THEN
        GVL_DISTRIBUTED_COMMIT.Peer_Commit_Mismatch := TRUE;

        L_Commit_Valid := FALSE;
        L_Error_Code := 15003;
        L_Error_Text := 'Peer commit epoch mismatch';
    END_IF;
END_IF;

IF L_Commit_Valid AND L_Peer_Session_Active THEN
    IF GVL_DISTRIBUTED_COMMIT.Peer_Prepare_Epoch < GVL_DISTRIBUTED_COMMIT.Local_Prepare_Epoch THEN
        GVL_DISTRIBUTED_COMMIT.Peer_Commit_Replay_Detected := TRUE;

        L_Commit_Valid := FALSE;
        L_Error_Code := 15004;
        L_Error_Text := 'Peer commit replay detected';
    END_IF;
END_IF;

IF L_Commit_Valid THEN
    GVL_DISTRIBUTED_COMMIT.Distributed_Commit_Epoch := GVL_DISTRIBUTED_COMMIT.Distributed_Commit_Epoch + 1;
    GVL_DISTRIBUTED_COMMIT.Distributed_Commit_Reconciliation_Epoch := GVL_DISTRIBUTED_COMMIT.Distributed_Commit_Reconciliation_Epoch + 1;

    GVL_DISTRIBUTED_COMMIT.Publication_Commit_Requested := TRUE;

    IF L_Peer_Session_Active THEN
        GVL_DISTRIBUTED_COMMIT.Publication_Commit_Confirmed := TRUE;
        GVL_DISTRIBUTED_COMMIT.Commit_Lease_Active := TRUE;
    ELSE
        GVL_DISTRIBUTED_COMMIT.Publication_Commit_Confirmed := FALSE;
        GVL_DISTRIBUTED_COMMIT.Commit_Lease_Active := FALSE;
    END_IF;

    GVL_DISTRIBUTED_COMMIT.Distributed_Commit_Valid := TRUE;

    IF GVL_CONVERGENCE.Convergence_Release_Allowed THEN
        GVL_DISTRIBUTED_COMMIT.Distributed_Commit_Quarantine_Active := FALSE;
    END_IF;

    GVL_DISTRIBUTED_COMMIT.Commit_Last_Reconciliation_MS := L_Now_MS;

    GVL_DISTRIBUTED_COMMIT.Distributed_Commit_Last_Error_Code := 0;
    GVL_DISTRIBUTED_COMMIT.Distributed_Commit_Last_Error_Text := '';
ELSE
    GVL_DISTRIBUTED_COMMIT.Publication_Commit_Confirmed := FALSE;

    GVL_DISTRIBUTED_COMMIT.Distributed_Commit_Valid := FALSE;
    GVL_DISTRIBUTED_COMMIT.Distributed_Commit_Quarantine_Active := TRUE;

    GVL_DISTRIBUTED_COMMIT.Distributed_Commit_Last_Error_Code := L_Error_Code;
    GVL_DISTRIBUTED_COMMIT.Distributed_Commit_Last_Error_Text := L_Error_Text;
END_IF;
END_PROGRAM

(* ---- PRG_Distributed_Safety_Reality_Consensus_Governor.st ---- *)
PROGRAM PRG_Distributed_Safety_Reality_Consensus_Governor
IF GVL_UNSAFE_TRANSITION_FORENSICS_FABRIC.Unsafe_Transition_Forensics_Granted
AND NOT GVL_DISTRIBUTED_SAFETY_REALITY_CONSENSUS_FABRIC.Distributed_Safety_State_Fork
AND NOT GVL_DISTRIBUTED_SAFETY_REALITY_CONSENSUS_FABRIC.Cluster_Safety_Projection_Drift
AND NOT GVL_DISTRIBUTED_SAFETY_REALITY_CONSENSUS_FABRIC.Distributed_Unsafe_State_Hidden THEN

    GVL_DISTRIBUTED_SAFETY_REALITY_CONSENSUS_FABRIC.Distributed_Safety_Reality_Consensus_Valid := TRUE;
    GVL_DISTRIBUTED_SAFETY_REALITY_CONSENSUS_FABRIC.Distributed_Safety_Reality_Consensus_Granted := TRUE;
    GVL_DISTRIBUTED_SAFETY_REALITY_CONSENSUS_FABRIC.Distributed_Safety_Consensus_Valid := TRUE;
    GVL_DISTRIBUTED_SAFETY_REALITY_CONSENSUS_FABRIC.Cluster_Safety_Reality_Stable := TRUE;
    GVL_DISTRIBUTED_SAFETY_REALITY_CONSENSUS_FABRIC.Distributed_Observability_Reality_Equivalence := TRUE;
END_IF;
END_PROGRAM

(* ---- PRG_Energy_Isolation_Causality_Governor.st ---- *)
PROGRAM PRG_Energy_Isolation_Causality_Governor
IF GVL_AUTHORITY_RESURRECTION_BOUNDARY_FABRIC.Authority_Resurrection_Boundary_Valid
AND NOT GVL_ENERGY_ISOLATION_CAUSALITY_FABRIC.Residual_Energy_Leakage_Detected
AND NOT GVL_ENERGY_ISOLATION_CAUSALITY_FABRIC.CrossDomain_Power_Backfeed_Detected
AND NOT GVL_ENERGY_ISOLATION_CAUSALITY_FABRIC.SplitEnergy_Topology_Detected
AND NOT GVL_ENERGY_ISOLATION_CAUSALITY_FABRIC.Unsafe_Energy_Propagation_Detected THEN

    GVL_ENERGY_ISOLATION_CAUSALITY_FABRIC.Energy_Isolation_Causality_Valid := TRUE;
    GVL_ENERGY_ISOLATION_CAUSALITY_FABRIC.Energy_Isolation_Causality_Granted := TRUE;
    GVL_ENERGY_ISOLATION_CAUSALITY_FABRIC.Physical_Energy_Isolation_Valid := TRUE;
    GVL_ENERGY_ISOLATION_CAUSALITY_FABRIC.Unsafe_Energy_Propagation_Prevented := TRUE;
    GVL_ENERGY_ISOLATION_CAUSALITY_FABRIC.CrossDomain_Power_Segmentation_Canonical := TRUE;
END_IF;
END_PROGRAM

(* ---- PRG_Environmental_Authority_Governor.st ---- *)
PROGRAM PRG_Environmental_Authority_Governor
VAR
    L_Now_MS : UDINT;
    L_Environment_Valid : BOOL := TRUE;
    L_Error_Code : UDINT := 0;
    L_Error_Text : STRING(160) := '';
END_VAR

L_Now_MS := GVL_STATUS.G_System_Time_MS;
L_Environment_Valid := TRUE;
L_Error_Code := 0;
L_Error_Text := '';

// Fail-safe defaults.
GVL_ENVIRONMENTAL_AUTHORITY.Environmental_Authority_Valid := FALSE;
GVL_ENVIRONMENTAL_AUTHORITY.Environmental_Authority_Granted := FALSE;
GVL_ENVIRONMENTAL_AUTHORITY.Environmental_Quarantine_Active := TRUE;

GVL_ENVIRONMENTAL_AUTHORITY.External_Environment_Causally_Compatible := FALSE;
GVL_ENVIRONMENTAL_AUTHORITY.Utility_Environment_Stable := FALSE;
GVL_ENVIRONMENTAL_AUTHORITY.Hydraulic_Source_Stable := FALSE;
GVL_ENVIRONMENTAL_AUTHORITY.Thermal_Environment_Stable := FALSE;
GVL_ENVIRONMENTAL_AUTHORITY.Airflow_Environment_Stable := FALSE;

// Environmental authority requires temporal stability.
IF NOT GVL_TEMPORAL_STABILITY.Temporal_Stability_Granted THEN
    L_Environment_Valid := FALSE;
    L_Error_Code := 29000;
    L_Error_Text := 'Temporal stability authority not granted';
END_IF;

// Freeze propagation detection.
IF GVL_ENVIRONMENTAL_AUTHORITY.Freeze_Front_Propagation_Detected THEN
    L_Environment_Valid := FALSE;
    L_Error_Code := 29001;
    L_Error_Text := 'Freeze-front propagation detected';
END_IF;

// Utility instability propagation.
IF GVL_ENVIRONMENTAL_AUTHORITY.Utility_Instability_Propagation_Detected THEN
    L_Environment_Valid := FALSE;
    L_Error_Code := 29002;
    L_Error_Text := 'Utility instability propagation detected';
END_IF;

// Hydraulic collapse prediction.
IF GVL_ENVIRONMENTAL_AUTHORITY.External_Hydraulic_Collapse_Detected THEN
    L_Environment_Valid := FALSE;
    L_Error_Code := 29003;
    L_Error_Text := 'External hydraulic collapse detected';
END_IF;

// Airflow icing conditions.
IF GVL_ENVIRONMENTAL_AUTHORITY.Airflow_Icing_Condition_Detected THEN
    L_Environment_Valid := FALSE;
    L_Error_Code := 29004;
    L_Error_Text := 'Airflow icing condition detected';
END_IF;

// Environmental rebound race.
IF GVL_ENVIRONMENTAL_AUTHORITY.Environmental_Rebound_Race_Detected THEN
    L_Environment_Valid := FALSE;
    L_Error_Code := 29005;
    L_Error_Text := 'Environmental rebound race detected';
END_IF;

// External environment validation.
IF L_Environment_Valid
AND NOT GVL_ENVIRONMENTAL_AUTHORITY.Mains_Quality_Valid THEN
    L_Environment_Valid := FALSE;
    L_Error_Code := 29010;
    L_Error_Text := 'Mains quality invalid';
END_IF;

IF L_Environment_Valid
AND NOT GVL_ENVIRONMENTAL_AUTHORITY.Supply_Water_Available THEN
    L_Environment_Valid := FALSE;
    L_Error_Code := 29011;
    L_Error_Text := 'Supply water unavailable';
END_IF;

IF L_Environment_Valid
AND NOT GVL_ENVIRONMENTAL_AUTHORITY.Outdoor_Airflow_Valid THEN
    L_Environment_Valid := FALSE;
    L_Error_Code := 29012;
    L_Error_Text := 'Outdoor airflow invalid';
END_IF;

IF L_Environment_Valid
AND NOT GVL_ENVIRONMENTAL_AUTHORITY.Freeze_Protection_Valid THEN
    L_Environment_Valid := FALSE;
    L_Error_Code := 29013;
    L_Error_Text := 'Freeze protection invalid';
END_IF;

IF L_Environment_Valid THEN
    GVL_ENVIRONMENTAL_AUTHORITY.Environmental_Authority_Valid := TRUE;
    GVL_ENVIRONMENTAL_AUTHORITY.Environmental_Authority_Granted := TRUE;
    GVL_ENVIRONMENTAL_AUTHORITY.Environmental_Quarantine_Active := FALSE;

    GVL_ENVIRONMENTAL_AUTHORITY.External_Environment_Causally_Compatible := TRUE;
    GVL_ENVIRONMENTAL_AUTHORITY.Utility_Environment_Stable := TRUE;
    GVL_ENVIRONMENTAL_AUTHORITY.Hydraulic_Source_Stable := TRUE;
    GVL_ENVIRONMENTAL_AUTHORITY.Thermal_Environment_Stable := TRUE;
    GVL_ENVIRONMENTAL_AUTHORITY.Airflow_Environment_Stable := TRUE;

    GVL_ENVIRONMENTAL_AUTHORITY.Environmental_Authority_Epoch :=
        GVL_TEMPORAL_STABILITY.Temporal_Stability_Epoch;

    GVL_ENVIRONMENTAL_AUTHORITY.Environmental_Authority_Epoch_Coherent := TRUE;

    GVL_ENVIRONMENTAL_AUTHORITY.Environmental_Last_Update_MS :=
        L_Now_MS;

    GVL_ENVIRONMENTAL_AUTHORITY.Environmental_Lease_Expired := FALSE;

    GVL_ENVIRONMENTAL_AUTHORITY.Environmental_Last_Error_Code := 0;
    GVL_ENVIRONMENTAL_AUTHORITY.Environmental_Last_Error_Text := '';
ELSE
    GVL_ENVIRONMENTAL_AUTHORITY.Environmental_Authority_Valid := FALSE;
    GVL_ENVIRONMENTAL_AUTHORITY.Environmental_Authority_Granted := FALSE;
    GVL_ENVIRONMENTAL_AUTHORITY.Environmental_Quarantine_Active := TRUE;

    GVL_ENVIRONMENTAL_AUTHORITY.Environmental_Lease_Expired := TRUE;

    GVL_ENVIRONMENTAL_AUTHORITY.Environmental_Last_Error_Code :=
        L_Error_Code;

    GVL_ENVIRONMENTAL_AUTHORITY.Environmental_Last_Error_Text :=
        L_Error_Text;

    GVL_ENVIRONMENTAL_AUTHORITY.Environmental_Invalidation_Count :=
        GVL_ENVIRONMENTAL_AUTHORITY.Environmental_Invalidation_Count + 1;
END_IF;

END_PROGRAM

(* ---- PRG_Execution_Projection_Integrity_Governor.st ---- *)
PROGRAM PRG_Execution_Projection_Integrity_Governor
VAR
    L_Now_MS : UDINT;
    L_Integrity_Valid : BOOL := TRUE;
    L_Error_Code : UDINT := 0;
    L_Error_Text : STRING(160) := '';
END_VAR

L_Now_MS := GVL_STATUS.G_System_Time_MS;
L_Integrity_Valid := TRUE;
L_Error_Code := 0;
L_Error_Text := '';

// Fail-safe defaults.
GVL_EXECUTION_PROJECTION_INTEGRITY_FABRIC.Execution_Projection_Integrity_Valid := FALSE;
GVL_EXECUTION_PROJECTION_INTEGRITY_FABRIC.Execution_Projection_Integrity_Granted := FALSE;
GVL_EXECUTION_PROJECTION_INTEGRITY_FABRIC.Execution_Projection_Integrity_Quarantine_Active := TRUE;

GVL_EXECUTION_PROJECTION_INTEGRITY_FABRIC.Execution_Authority_Projection_Consistent := FALSE;
GVL_EXECUTION_PROJECTION_INTEGRITY_FABRIC.CrossDomain_Actuation_Enforcement_Aligned := FALSE;
GVL_EXECUTION_PROJECTION_INTEGRITY_FABRIC.Physical_Execution_Governance_Canonical := FALSE;
GVL_EXECUTION_PROJECTION_INTEGRITY_FABRIC.Actuation_Surface_Consensus_Valid := FALSE;
GVL_EXECUTION_PROJECTION_INTEGRITY_FABRIC.Execution_Projection_Lineage_Coherent := FALSE;

// Governance observer consensus required.
IF NOT GVL_GOVERNANCE_OBSERVER_CONSENSUS_FABRIC.Governance_Observer_Consensus_Granted THEN
    L_Integrity_Valid := FALSE;
    L_Error_Code := 51000;
    L_Error_Text := 'Governance observer consensus not granted';
END_IF;

// Execution projection split-brain detectors.
IF GVL_EXECUTION_PROJECTION_INTEGRITY_FABRIC.Execution_Projection_Divergence_Detected THEN
    L_Integrity_Valid := FALSE;
    L_Error_Code := 51001;
    L_Error_Text := 'Execution projection divergence detected';
END_IF;

IF GVL_EXECUTION_PROJECTION_INTEGRITY_FABRIC.Actuation_Path_Authority_Bypass_Detected THEN
    L_Integrity_Valid := FALSE;
    L_Error_Code := 51002;
    L_Error_Text := 'Actuation path authority bypass detected';
END_IF;

IF GVL_EXECUTION_PROJECTION_INTEGRITY_FABRIC.CrossDomain_Enforcement_Fork_Detected THEN
    L_Integrity_Valid := FALSE;
    L_Error_Code := 51003;
    L_Error_Text := 'Cross-domain enforcement fork detected';
END_IF;

IF GVL_EXECUTION_PROJECTION_INTEGRITY_FABRIC.Canonical_Governance_Execution_Lost THEN
    L_Integrity_Valid := FALSE;
    L_Error_Code := 51004;
    L_Error_Text := 'Canonical governance execution lost';
END_IF;

IF GVL_EXECUTION_PROJECTION_INTEGRITY_FABRIC.Runtime_Execution_Lineage_Drift_Detected THEN
    L_Integrity_Valid := FALSE;
    L_Error_Code := 51005;
    L_Error_Text := 'Runtime execution lineage drift detected';
END_IF;

IF GVL_EXECUTION_PROJECTION_INTEGRITY_FABRIC.Distributed_Actuation_Reality_Fork_Detected THEN
    L_Integrity_Valid := FALSE;
    L_Error_Code := 51006;
    L_Error_Text := 'Distributed actuation reality fork detected';
END_IF;

// Execution enforcement validation.
IF L_Integrity_Valid
AND NOT GVL_EXECUTION_PROJECTION_INTEGRITY_FABRIC.Runtime_Actuation_Projection_Stable THEN
    L_Integrity_Valid := FALSE;
    L_Error_Code := 51010;
    L_Error_Text := 'Runtime actuation projection invalid';
END_IF;

IF L_Integrity_Valid
AND NOT GVL_EXECUTION_PROJECTION_INTEGRITY_FABRIC.Distributed_Execution_Equivalence_Valid THEN
    L_Integrity_Valid := FALSE;
    L_Error_Code := 51011;
    L_Error_Text := 'Distributed execution equivalence invalid';
END_IF;

IF L_Integrity_Valid
AND NOT GVL_EXECUTION_PROJECTION_INTEGRITY_FABRIC.Execution_Governance_Causality_Grounded THEN
    L_Integrity_Valid := FALSE;
    L_Error_Code := 51012;
    L_Error_Text := 'Execution governance causality invalid';
END_IF;

IF L_Integrity_Valid
AND NOT GVL_EXECUTION_PROJECTION_INTEGRITY_FABRIC.Physical_Enforcement_Timeline_Monotonic THEN
    L_Integrity_Valid := FALSE;
    L_Error_Code := 51013;
    L_Error_Text := 'Physical enforcement timeline monotonicity invalid';
END_IF;

IF L_Integrity_Valid THEN
    GVL_EXECUTION_PROJECTION_INTEGRITY_FABRIC.Execution_Projection_Integrity_Valid := TRUE;
    GVL_EXECUTION_PROJECTION_INTEGRITY_FABRIC.Execution_Projection_Integrity_Granted := TRUE;
    GVL_EXECUTION_PROJECTION_INTEGRITY_FABRIC.Execution_Projection_Integrity_Quarantine_Active := FALSE;

    GVL_EXECUTION_PROJECTION_INTEGRITY_FABRIC.Execution_Authority_Projection_Consistent := TRUE;
    GVL_EXECUTION_PROJECTION_INTEGRITY_FABRIC.CrossDomain_Actuation_Enforcement_Aligned := TRUE;
    GVL_EXECUTION_PROJECTION_INTEGRITY_FABRIC.Physical_Execution_Governance_Canonical := TRUE;
    GVL_EXECUTION_PROJECTION_INTEGRITY_FABRIC.Actuation_Surface_Consensus_Valid := TRUE;
    GVL_EXECUTION_PROJECTION_INTEGRITY_FABRIC.Execution_Projection_Lineage_Coherent := TRUE;

    GVL_EXECUTION_PROJECTION_INTEGRITY_FABRIC.Execution_Projection_Integrity_Epoch :=
        GVL_GOVERNANCE_OBSERVER_CONSENSUS_FABRIC.Governance_Observer_Consensus_Epoch;

    GVL_EXECUTION_PROJECTION_INTEGRITY_FABRIC.Execution_Projection_Integrity_Epoch_Coherent := TRUE;

    GVL_EXECUTION_PROJECTION_INTEGRITY_FABRIC.Execution_Projection_Integrity_Last_Update_MS :=
        L_Now_MS;

    GVL_EXECUTION_PROJECTION_INTEGRITY_FABRIC.Execution_Projection_Integrity_Lease_Expired := FALSE;

    GVL_EXECUTION_PROJECTION_INTEGRITY_FABRIC.Execution_Projection_Integrity_Last_Error_Code := 0;
    GVL_EXECUTION_PROJECTION_INTEGRITY_FABRIC.Execution_Projection_Integrity_Last_Error_Text := '';
ELSE
    GVL_EXECUTION_PROJECTION_INTEGRITY_FABRIC.Execution_Projection_Integrity_Valid := FALSE;
    GVL_EXECUTION_PROJECTION_INTEGRITY_FABRIC.Execution_Projection_Integrity_Granted := FALSE;
    GVL_EXECUTION_PROJECTION_INTEGRITY_FABRIC.Execution_Projection_Integrity_Quarantine_Active := TRUE;

    GVL_EXECUTION_PROJECTION_INTEGRITY_FABRIC.Execution_Projection_Integrity_Lease_Expired := TRUE;

    GVL_EXECUTION_PROJECTION_INTEGRITY_FABRIC.Execution_Projection_Integrity_Last_Error_Code :=
        L_Error_Code;

    GVL_EXECUTION_PROJECTION_INTEGRITY_FABRIC.Execution_Projection_Integrity_Last_Error_Text :=
        L_Error_Text;

    GVL_EXECUTION_PROJECTION_INTEGRITY_FABRIC.Execution_Projection_Integrity_Invalidation_Count :=
        GVL_EXECUTION_PROJECTION_INTEGRITY_FABRIC.Execution_Projection_Integrity_Invalidation_Count + 1;
END_IF;

END_PROGRAM

(* ---- PRG_Global_Authority_Sync_Governor.st ---- *)
PROGRAM PRG_Global_Authority_Sync_Governor
VAR
    L_Now_MS : UDINT;
    L_Global_Valid : BOOL := TRUE;
    L_Error_Code : UDINT := 0;
    L_Error_Text : STRING(160) := '';
END_VAR

L_Now_MS := GVL_STATUS.G_System_Time_MS;
L_Global_Valid := TRUE;
L_Error_Code := 0;
L_Error_Text := '';

// Fail-safe defaults.
GVL_GLOBAL_AUTHORITY_SYNC.Global_Authority_Sync_Valid := FALSE;
GVL_GLOBAL_AUTHORITY_SYNC.Global_Authority_Sync_Granted := FALSE;
GVL_GLOBAL_AUTHORITY_SYNC.Global_Authority_Sync_Quarantine_Active := TRUE;

GVL_GLOBAL_AUTHORITY_SYNC.Heating_Authority_Coherent := FALSE;
GVL_GLOBAL_AUTHORITY_SYNC.Ventilation_Authority_Coherent := FALSE;
GVL_GLOBAL_AUTHORITY_SYNC.Water_Authority_Coherent := FALSE;
GVL_GLOBAL_AUTHORITY_SYNC.Access_Authority_Coherent := FALSE;
GVL_GLOBAL_AUTHORITY_SYNC.Lighting_Authority_Coherent := FALSE;

// Historical truth authority required.
IF NOT GVL_HISTORICAL_TRUTH.Historical_Truth_Granted THEN
    L_Global_Valid := FALSE;
    L_Error_Code := 34000;
    L_Error_Text := 'Historical truth authority not granted';
END_IF;

// Cross-domain split-brain detectors.
IF GVL_GLOBAL_AUTHORITY_SYNC.Authority_Epoch_Fragmentation_Detected THEN
    L_Global_Valid := FALSE;
    L_Error_Code := 34001;
    L_Error_Text := 'Authority epoch fragmentation detected';
END_IF;

IF GVL_GLOBAL_AUTHORITY_SYNC.Partial_Recovery_SplitBrain_Detected THEN
    L_Global_Valid := FALSE;
    L_Error_Code := 34002;
    L_Error_Text := 'Partial recovery split-brain detected';
END_IF;

IF GVL_GLOBAL_AUTHORITY_SYNC.Cross_Domain_Replay_Skew_Detected THEN
    L_Global_Valid := FALSE;
    L_Error_Code := 34003;
    L_Error_Text := 'Cross-domain replay skew detected';
END_IF;

IF GVL_GLOBAL_AUTHORITY_SYNC.Distributed_Authority_Divergence_Detected THEN
    L_Global_Valid := FALSE;
    L_Error_Code := 34004;
    L_Error_Text := 'Distributed authority divergence detected';
END_IF;

IF GVL_GLOBAL_AUTHORITY_SYNC.Global_Causality_Desynchronization_Detected THEN
    L_Global_Valid := FALSE;
    L_Error_Code := 34005;
    L_Error_Text := 'Global causality desynchronization detected';
END_IF;

IF GVL_GLOBAL_AUTHORITY_SYNC.Multi_Domain_Chronology_Drift_Detected THEN
    L_Global_Valid := FALSE;
    L_Error_Code := 34006;
    L_Error_Text := 'Multi-domain chronology drift detected';
END_IF;

// Cross-domain synchronization validation.
IF L_Global_Valid
AND NOT GVL_GLOBAL_AUTHORITY_SYNC.Cross_Domain_Epoch_Coherent THEN
    L_Global_Valid := FALSE;
    L_Error_Code := 34010;
    L_Error_Text := 'Cross-domain epoch coherence invalid';
END_IF;

IF L_Global_Valid
AND NOT GVL_GLOBAL_AUTHORITY_SYNC.Distributed_Authority_Generation_Coherent THEN
    L_Global_Valid := FALSE;
    L_Error_Code := 34011;
    L_Error_Text := 'Distributed authority generation coherence invalid';
END_IF;

IF L_Global_Valid
AND NOT GVL_GLOBAL_AUTHORITY_SYNC.Global_Causality_Timeline_Stable THEN
    L_Global_Valid := FALSE;
    L_Error_Code := 34012;
    L_Error_Text := 'Global causality timeline unstable';
END_IF;

IF L_Global_Valid
AND NOT GVL_GLOBAL_AUTHORITY_SYNC.Multi_Domain_Recovery_Coherent THEN
    L_Global_Valid := FALSE;
    L_Error_Code := 34013;
    L_Error_Text := 'Multi-domain recovery coherence invalid';
END_IF;

IF L_Global_Valid THEN
    GVL_GLOBAL_AUTHORITY_SYNC.Global_Authority_Sync_Valid := TRUE;
    GVL_GLOBAL_AUTHORITY_SYNC.Global_Authority_Sync_Granted := TRUE;
    GVL_GLOBAL_AUTHORITY_SYNC.Global_Authority_Sync_Quarantine_Active := FALSE;

    GVL_GLOBAL_AUTHORITY_SYNC.Heating_Authority_Coherent := TRUE;
    GVL_GLOBAL_AUTHORITY_SYNC.Ventilation_Authority_Coherent := TRUE;
    GVL_GLOBAL_AUTHORITY_SYNC.Water_Authority_Coherent := TRUE;
    GVL_GLOBAL_AUTHORITY_SYNC.Access_Authority_Coherent := TRUE;
    GVL_GLOBAL_AUTHORITY_SYNC.Lighting_Authority_Coherent := TRUE;

    GVL_GLOBAL_AUTHORITY_SYNC.Global_Authority_Epoch :=
        GVL_HISTORICAL_TRUTH.Historical_Truth_Epoch;

    GVL_GLOBAL_AUTHORITY_SYNC.Global_Authority_Epoch_Coherent := TRUE;

    GVL_GLOBAL_AUTHORITY_SYNC.Global_Authority_Last_Update_MS := L_Now_MS;
    GVL_GLOBAL_AUTHORITY_SYNC.Global_Authority_Lease_Expired := FALSE;

    GVL_GLOBAL_AUTHORITY_SYNC.Global_Authority_Last_Error_Code := 0;
    GVL_GLOBAL_AUTHORITY_SYNC.Global_Authority_Last_Error_Text := '';
ELSE
    GVL_GLOBAL_AUTHORITY_SYNC.Global_Authority_Sync_Valid := FALSE;
    GVL_GLOBAL_AUTHORITY_SYNC.Global_Authority_Sync_Granted := FALSE;
    GVL_GLOBAL_AUTHORITY_SYNC.Global_Authority_Sync_Quarantine_Active := TRUE;

    GVL_GLOBAL_AUTHORITY_SYNC.Global_Authority_Lease_Expired := TRUE;

    GVL_GLOBAL_AUTHORITY_SYNC.Global_Authority_Last_Error_Code :=
        L_Error_Code;

    GVL_GLOBAL_AUTHORITY_SYNC.Global_Authority_Last_Error_Text :=
        L_Error_Text;

    GVL_GLOBAL_AUTHORITY_SYNC.Global_Authority_Invalidation_Count :=
        GVL_GLOBAL_AUTHORITY_SYNC.Global_Authority_Invalidation_Count + 1;
END_IF;

END_PROGRAM

(* ---- PRG_Governance_Feedback_Integrity_Governor.st ---- *)
PROGRAM PRG_Governance_Feedback_Integrity_Governor
VAR
    L_Now_MS : UDINT;
    L_Integrity_Valid : BOOL := TRUE;
    L_Error_Code : UDINT := 0;
    L_Error_Text : STRING(160) := '';
END_VAR

L_Now_MS := GVL_STATUS.G_System_Time_MS;
L_Integrity_Valid := TRUE;
L_Error_Code := 0;
L_Error_Text := '';

// Fail-safe defaults.
GVL_GOVERNANCE_FEEDBACK_INTEGRITY_FABRIC.Governance_Feedback_Integrity_Valid := FALSE;
GVL_GOVERNANCE_FEEDBACK_INTEGRITY_FABRIC.Governance_Feedback_Integrity_Granted := FALSE;
GVL_GOVERNANCE_FEEDBACK_INTEGRITY_FABRIC.Governance_Feedback_Integrity_Quarantine_Active := TRUE;

GVL_GOVERNANCE_FEEDBACK_INTEGRITY_FABRIC.Execution_Feedback_Causality_Isolated := FALSE;
GVL_GOVERNANCE_FEEDBACK_INTEGRITY_FABRIC.Governance_Derivation_Inputs_Canonical := FALSE;
GVL_GOVERNANCE_FEEDBACK_INTEGRITY_FABRIC.Telemetry_To_Authority_Lineage_Valid := FALSE;
GVL_GOVERNANCE_FEEDBACK_INTEGRITY_FABRIC.Feedback_Epoch_Integrity_Stable := FALSE;
GVL_GOVERNANCE_FEEDBACK_INTEGRITY_FABRIC.Governance_Feedback_Lineage_Coherent := FALSE;

// Execution projection integrity required.
IF NOT GVL_EXECUTION_PROJECTION_INTEGRITY_FABRIC.Execution_Projection_Integrity_Granted THEN
    L_Integrity_Valid := FALSE;
    L_Error_Code := 52000;
    L_Error_Text := 'Execution projection integrity not granted';
END_IF;

// Governance feedback poisoning detectors.
IF GVL_GOVERNANCE_FEEDBACK_INTEGRITY_FABRIC.Governance_Feedback_Poisoning_Detected THEN
    L_Integrity_Valid := FALSE;
    L_Error_Code := 52001;
    L_Error_Text := 'Governance feedback poisoning detected';
END_IF;

IF GVL_GOVERNANCE_FEEDBACK_INTEGRITY_FABRIC.Execution_Telemetry_Authority_Corruption THEN
    L_Integrity_Valid := FALSE;
    L_Error_Code := 52002;
    L_Error_Text := 'Execution telemetry authority corruption detected';
END_IF;

IF GVL_GOVERNANCE_FEEDBACK_INTEGRITY_FABRIC.CrossEpoch_Feedback_Lineage_Drift THEN
    L_Integrity_Valid := FALSE;
    L_Error_Code := 52003;
    L_Error_Text := 'Cross-epoch feedback lineage drift detected';
END_IF;

IF GVL_GOVERNANCE_FEEDBACK_INTEGRITY_FABRIC.Retroactive_Governance_Mutation_Detected THEN
    L_Integrity_Valid := FALSE;
    L_Error_Code := 52004;
    L_Error_Text := 'Retroactive governance mutation detected';
END_IF;

IF GVL_GOVERNANCE_FEEDBACK_INTEGRITY_FABRIC.Distributed_Feedback_Fork_Detected THEN
    L_Integrity_Valid := FALSE;
    L_Error_Code := 52005;
    L_Error_Text := 'Distributed feedback fork detected';
END_IF;

IF GVL_GOVERNANCE_FEEDBACK_INTEGRITY_FABRIC.Untrusted_Execution_Observation_Injected THEN
    L_Integrity_Valid := FALSE;
    L_Error_Code := 52006;
    L_Error_Text := 'Untrusted execution observation injected';
END_IF;

// Governance feedback validation.
IF L_Integrity_Valid
AND NOT GVL_GOVERNANCE_FEEDBACK_INTEGRITY_FABRIC.Authenticated_Execution_Observation_Valid THEN
    L_Integrity_Valid := FALSE;
    L_Error_Code := 52010;
    L_Error_Text := 'Authenticated execution observation invalid';
END_IF;

IF L_Integrity_Valid
AND NOT GVL_GOVERNANCE_FEEDBACK_INTEGRITY_FABRIC.CrossEpoch_Feedback_Continuity_Stable THEN
    L_Integrity_Valid := FALSE;
    L_Error_Code := 52011;
    L_Error_Text := 'Cross-epoch feedback continuity invalid';
END_IF;

IF L_Integrity_Valid
AND NOT GVL_GOVERNANCE_FEEDBACK_INTEGRITY_FABRIC.Governance_Input_Causality_Grounded THEN
    L_Integrity_Valid := FALSE;
    L_Error_Code := 52012;
    L_Error_Text := 'Governance input causality invalid';
END_IF;

IF L_Integrity_Valid
AND NOT GVL_GOVERNANCE_FEEDBACK_INTEGRITY_FABRIC.Distributed_Feedback_Consensus_Valid THEN
    L_Integrity_Valid := FALSE;
    L_Error_Code := 52013;
    L_Error_Text := 'Distributed feedback consensus invalid';
END_IF;

IF L_Integrity_Valid THEN
    GVL_GOVERNANCE_FEEDBACK_INTEGRITY_FABRIC.Governance_Feedback_Integrity_Valid := TRUE;
    GVL_GOVERNANCE_FEEDBACK_INTEGRITY_FABRIC.Governance_Feedback_Integrity_Granted := TRUE;
    GVL_GOVERNANCE_FEEDBACK_INTEGRITY_FABRIC.Governance_Feedback_Integrity_Quarantine_Active := FALSE;

    GVL_GOVERNANCE_FEEDBACK_INTEGRITY_FABRIC.Execution_Feedback_Causality_Isolated := TRUE;
    GVL_GOVERNANCE_FEEDBACK_INTEGRITY_FABRIC.Governance_Derivation_Inputs_Canonical := TRUE;
    GVL_GOVERNANCE_FEEDBACK_INTEGRITY_FABRIC.Telemetry_To_Authority_Lineage_Valid := TRUE;
    GVL_GOVERNANCE_FEEDBACK_INTEGRITY_FABRIC.Feedback_Epoch_Integrity_Stable := TRUE;
    GVL_GOVERNANCE_FEEDBACK_INTEGRITY_FABRIC.Governance_Feedback_Lineage_Coherent := TRUE;

    GVL_GOVERNANCE_FEEDBACK_INTEGRITY_FABRIC.Governance_Feedback_Integrity_Epoch :=
        GVL_EXECUTION_PROJECTION_INTEGRITY_FABRIC.Execution_Projection_Integrity_Epoch;

    GVL_GOVERNANCE_FEEDBACK_INTEGRITY_FABRIC.Governance_Feedback_Integrity_Epoch_Coherent := TRUE;

    GVL_GOVERNANCE_FEEDBACK_INTEGRITY_FABRIC.Governance_Feedback_Integrity_Last_Update_MS :=
        L_Now_MS;

    GVL_GOVERNANCE_FEEDBACK_INTEGRITY_FABRIC.Governance_Feedback_Integrity_Lease_Expired := FALSE;

    GVL_GOVERNANCE_FEEDBACK_INTEGRITY_FABRIC.Governance_Feedback_Integrity_Last_Error_Code := 0;
    GVL_GOVERNANCE_FEEDBACK_INTEGRITY_FABRIC.Governance_Feedback_Integrity_Last_Error_Text := '';
ELSE
    GVL_GOVERNANCE_FEEDBACK_INTEGRITY_FABRIC.Governance_Feedback_Integrity_Valid := FALSE;
    GVL_GOVERNANCE_FEEDBACK_INTEGRITY_FABRIC.Governance_Feedback_Integrity_Granted := FALSE;
    GVL_GOVERNANCE_FEEDBACK_INTEGRITY_FABRIC.Governance_Feedback_Integrity_Quarantine_Active := TRUE;

    GVL_GOVERNANCE_FEEDBACK_INTEGRITY_FABRIC.Governance_Feedback_Integrity_Lease_Expired := TRUE;

    GVL_GOVERNANCE_FEEDBACK_INTEGRITY_FABRIC.Governance_Feedback_Integrity_Last_Error_Code :=
        L_Error_Code;

    GVL_GOVERNANCE_FEEDBACK_INTEGRITY_FABRIC.Governance_Feedback_Integrity_Last_Error_Text :=
        L_Error_Text;

    GVL_GOVERNANCE_FEEDBACK_INTEGRITY_FABRIC.Governance_Feedback_Integrity_Invalidation_Count :=
        GVL_GOVERNANCE_FEEDBACK_INTEGRITY_FABRIC.Governance_Feedback_Integrity_Invalidation_Count + 1;
END_IF;

END_PROGRAM

(* ---- PRG_Governance_Validator_Integrity_Governor.st ---- *)
PROGRAM PRG_Governance_Validator_Integrity_Governor
VAR
    L_Now_MS : UDINT;
    L_Integrity_Valid : BOOL := TRUE;
    L_Error_Code : UDINT := 0;
    L_Error_Text : STRING(160) := '';
END_VAR

L_Now_MS := GVL_STATUS.G_System_Time_MS;
L_Integrity_Valid := TRUE;
L_Error_Code := 0;
L_Error_Text := '';

// Fail-safe defaults.
GVL_GOVERNANCE_VALIDATOR_INTEGRITY_FABRIC.Governance_Validator_Integrity_Valid := FALSE;
GVL_GOVERNANCE_VALIDATOR_INTEGRITY_FABRIC.Governance_Validator_Integrity_Granted := FALSE;
GVL_GOVERNANCE_VALIDATOR_INTEGRITY_FABRIC.Governance_Validator_Integrity_Quarantine_Active := TRUE;

GVL_GOVERNANCE_VALIDATOR_INTEGRITY_FABRIC.Validator_Semantics_Immutable := FALSE;
GVL_GOVERNANCE_VALIDATOR_INTEGRITY_FABRIC.CrossEpoch_Validation_Equivalence_Stable := FALSE;
GVL_GOVERNANCE_VALIDATOR_INTEGRITY_FABRIC.Distributed_Validator_Consensus_Valid := FALSE;
GVL_GOVERNANCE_VALIDATOR_INTEGRITY_FABRIC.Governance_Rule_Integrity_Canonical := FALSE;
GVL_GOVERNANCE_VALIDATOR_INTEGRITY_FABRIC.Validator_Lineage_Coherent := FALSE;

// Governance feedback integrity required.
IF NOT GVL_GOVERNANCE_FEEDBACK_INTEGRITY_FABRIC.Governance_Feedback_Integrity_Granted THEN
    L_Integrity_Valid := FALSE;
    L_Error_Code := 53000;
    L_Error_Text := 'Governance feedback integrity not granted';
END_IF;

// Validator self-corruption detectors.
IF GVL_GOVERNANCE_VALIDATOR_INTEGRITY_FABRIC.Validator_Semantic_Drift_Detected THEN
    L_Integrity_Valid := FALSE;
    L_Error_Code := 53001;
    L_Error_Text := 'Validator semantic drift detected';
END_IF;

IF GVL_GOVERNANCE_VALIDATOR_INTEGRITY_FABRIC.CrossNode_Validation_Fork THEN
    L_Integrity_Valid := FALSE;
    L_Error_Code := 53002;
    L_Error_Text := 'Cross-node validation fork detected';
END_IF;

IF GVL_GOVERNANCE_VALIDATOR_INTEGRITY_FABRIC.Governance_Rule_Mutation_Detected THEN
    L_Integrity_Valid := FALSE;
    L_Error_Code := 53003;
    L_Error_Text := 'Governance rule mutation detected';
END_IF;

IF GVL_GOVERNANCE_VALIDATOR_INTEGRITY_FABRIC.SelfReferential_Validator_Corruption THEN
    L_Integrity_Valid := FALSE;
    L_Error_Code := 53004;
    L_Error_Text := 'Self-referential validator corruption detected';
END_IF;

IF GVL_GOVERNANCE_VALIDATOR_INTEGRITY_FABRIC.Validator_Lineage_Drift_Detected THEN
    L_Integrity_Valid := FALSE;
    L_Error_Code := 53005;
    L_Error_Text := 'Validator lineage drift detected';
END_IF;

IF GVL_GOVERNANCE_VALIDATOR_INTEGRITY_FABRIC.Distributed_Validator_Reality_Fork_Detected THEN
    L_Integrity_Valid := FALSE;
    L_Error_Code := 53006;
    L_Error_Text := 'Distributed validator reality fork detected';
END_IF;

// Validator integrity validation.
IF L_Integrity_Valid
AND NOT GVL_GOVERNANCE_VALIDATOR_INTEGRITY_FABRIC.Validator_Causality_Grounded THEN
    L_Integrity_Valid := FALSE;
    L_Error_Code := 53010;
    L_Error_Text := 'Validator causality invalid';
END_IF;

IF L_Integrity_Valid
AND NOT GVL_GOVERNANCE_VALIDATOR_INTEGRITY_FABRIC.Governance_Rule_Evolution_Governed THEN
    L_Integrity_Valid := FALSE;
    L_Error_Code := 53011;
    L_Error_Text := 'Governance rule evolution invalid';
END_IF;

IF L_Integrity_Valid
AND NOT GVL_GOVERNANCE_VALIDATOR_INTEGRITY_FABRIC.Distributed_Validation_Timeline_Monotonic THEN
    L_Integrity_Valid := FALSE;
    L_Error_Code := 53012;
    L_Error_Text := 'Distributed validation timeline monotonicity invalid';
END_IF;

IF L_Integrity_Valid
AND NOT GVL_GOVERNANCE_VALIDATOR_INTEGRITY_FABRIC.Validator_Interpretation_Equivalence_Valid THEN
    L_Integrity_Valid := FALSE;
    L_Error_Code := 53013;
    L_Error_Text := 'Validator interpretation equivalence invalid';
END_IF;

IF L_Integrity_Valid THEN
    GVL_GOVERNANCE_VALIDATOR_INTEGRITY_FABRIC.Governance_Validator_Integrity_Valid := TRUE;
    GVL_GOVERNANCE_VALIDATOR_INTEGRITY_FABRIC.Governance_Validator_Integrity_Granted := TRUE;
    GVL_GOVERNANCE_VALIDATOR_INTEGRITY_FABRIC.Governance_Validator_Integrity_Quarantine_Active := FALSE;

    GVL_GOVERNANCE_VALIDATOR_INTEGRITY_FABRIC.Validator_Semantics_Immutable := TRUE;
    GVL_GOVERNANCE_VALIDATOR_INTEGRITY_FABRIC.CrossEpoch_Validation_Equivalence_Stable := TRUE;
    GVL_GOVERNANCE_VALIDATOR_INTEGRITY_FABRIC.Distributed_Validator_Consensus_Valid := TRUE;
    GVL_GOVERNANCE_VALIDATOR_INTEGRITY_FABRIC.Governance_Rule_Integrity_Canonical := TRUE;
    GVL_GOVERNANCE_VALIDATOR_INTEGRITY_FABRIC.Validator_Lineage_Coherent := TRUE;

    GVL_GOVERNANCE_VALIDATOR_INTEGRITY_FABRIC.Governance_Validator_Integrity_Epoch :=
        GVL_GOVERNANCE_FEEDBACK_INTEGRITY_FABRIC.Governance_Feedback_Integrity_Epoch;

    GVL_GOVERNANCE_VALIDATOR_INTEGRITY_FABRIC.Governance_Validator_Integrity_Epoch_Coherent := TRUE;

    GVL_GOVERNANCE_VALIDATOR_INTEGRITY_FABRIC.Governance_Validator_Integrity_Last_Update_MS :=
        L_Now_MS;

    GVL_GOVERNANCE_VALIDATOR_INTEGRITY_FABRIC.Governance_Validator_Integrity_Lease_Expired := FALSE;

    GVL_GOVERNANCE_VALIDATOR_INTEGRITY_FABRIC.Governance_Validator_Integrity_Last_Error_Code := 0;
    GVL_GOVERNANCE_VALIDATOR_INTEGRITY_FABRIC.Governance_Validator_Integrity_Last_Error_Text := '';
ELSE
    GVL_GOVERNANCE_VALIDATOR_INTEGRITY_FABRIC.Governance_Validator_Integrity_Valid := FALSE;
    GVL_GOVERNANCE_VALIDATOR_INTEGRITY_FABRIC.Governance_Validator_Integrity_Granted := FALSE;
    GVL_GOVERNANCE_VALIDATOR_INTEGRITY_FABRIC.Governance_Validator_Integrity_Quarantine_Active := TRUE;

    GVL_GOVERNANCE_VALIDATOR_INTEGRITY_FABRIC.Governance_Validator_Integrity_Lease_Expired := TRUE;

    GVL_GOVERNANCE_VALIDATOR_INTEGRITY_FABRIC.Governance_Validator_Integrity_Last_Error_Code :=
        L_Error_Code;

    GVL_GOVERNANCE_VALIDATOR_INTEGRITY_FABRIC.Governance_Validator_Integrity_Last_Error_Text :=
        L_Error_Text;

    GVL_GOVERNANCE_VALIDATOR_INTEGRITY_FABRIC.Governance_Validator_Integrity_Invalidation_Count :=
        GVL_GOVERNANCE_VALIDATOR_INTEGRITY_FABRIC.Governance_Validator_Integrity_Invalidation_Count + 1;
END_IF;

END_PROGRAM
